METHOD  M_STATE_EXECUTING
VAR_INPUT
END_VAR
VAR_INST
	TargetLayer : INT;
	TargetSlide :E_WareHouseSlide;
END_VAR
VAR
	them: INT;
END_VAR
// Set FB state is busy
Busy := TRUE;

// Process
CASE uiExecutingStep OF
    0: // Command analize
		Ton_BoxMoveForward.IN := FALSE;
		Ton_ArriveDelay.IN := FALSE;
		tonFirstReserveTime.IN :=FALSE;
		tonSecondForwardTime.IN :=FALSE;
		tonThirdReserceTime.IN :=FALSE;
		TargetLayer := WarehouseCoordinates.Layer+(WarehouseSelect-1)*10 ; // Warehouse A=1 , B = 2;
		TargetSlide := WarehouseCoordinates.Slide;
		uiExecutingStep := 10;
		
	10:	//Motor reverse make sure have space can retreat
		Motors.arMotor[TargetLayer].M_MoveBackward();
		Ton_BoxMoveForward.IN := TRUE;
		IF NOT Motors.arMotor[TargetLayer].InStopped  THEN 
			uiExecutingStep := 15;
		END_IF
		IF Ton_BoxMoveForward.Q THEN
			_Error :=TRUE;
			Status :='Storage Cabinet MoveBackward motor timeout';
		END_IF
	15:	//Motor First reverse  then stop motor 
		tonFirstReserveTime.IN := TRUE;
		Ton_BoxMoveForward.IN := FALSE;
		IF tonFirstReserveTime.Q THEN
			tonFirstReserveTime.IN :=FALSE;
			Motors.arMotor[TargetLayer].M_MotorStop();// .M_MotorStop();//('FeedIn Motors.arMotor stop reverse');
			IF Motors.arMotor[TargetLayer].InStopped THEN
				uiExecutingStep := 20;
			END_IF
		END_IF
		
	20:	//Motor SecondForward check cabinet layer have't full box inside 
		Motors.arMotor[TargetLayer].M_MoveForward();// .M_MoveForward();//('FeedIn box : make sure have space can feedIn');
		Ton_BoxMoveForward.IN :=TRUE;
		IF NOT Motors.arMotor[TargetLayer].InStopped THEN
			uiExecutingStep := 25;
		END_IF
		IF Ton_BoxMoveForward.Q THEN
			_Error :=TRUE;
			Status :='Storage Cabinet MoveForward motor timeout';
		END_IF
		
	25:	//Motor second MoveForward  then stop motor
		tonSecondForwardTime.IN := TRUE;
		Ton_BoxMoveForward.IN := FALSE;
		IF tonSecondForwardTime.Q THEN
			tonSecondForwardTime.IN :=FALSE;
			Motors.arMotor[TargetLayer].M_MotorStop();//('');
			IF Motors.arMotor[TargetLayer].InStopped THEN
				uiExecutingStep :=30;
			END_IF
		END_IF
		
	30:	//check layer haven't full box behind
		M_CheckSlideSensor(WarehouseSelect := WarehouseSelect, 
						   WarehouseCoordinates := WarehouseCoordinates,
						   SensorStatus=>CurrentTargetSensorStatus);
		IF NOT  CurrentTargetSensorStatus THEN
			uiExecutingStep :=50;
		ELSE
			_Error :=TRUE;
			Status :='Storage Cabinet Layer full box inside ,plaease remove box ';
		END_IF	
		
	50:
        Motors.arMotor[TargetLayer].M_MoveBackward();// .M_MoveBackward();// ('FeedIn box : conveyor move backward');
		Ton_BoxMoveForward.IN := TRUE;
		IF  NOT Motors.arMotor[TargetLayer].InStopped THEN
			Ton_BoxMoveForward.IN := FALSE;	
			uiExecutingStep := 100;
		END_IF		
		IF  Ton_BoxMoveForward.Q THEN
		  _Error := TRUE;
           Status := 'Move motor timeout';
		END_IF
		
    100: // Wait box arrived
		M_CheckSlideSensor(WarehouseSelect := WarehouseSelect, 
						   WarehouseCoordinates := WarehouseCoordinates,
						   SensorStatus=>CurrentTargetSensorStatus);
        IF NOT CurrentTargetSensorStatus THEN
            uiExecutingStep := 200;
        END_IF
    200:// third reverse 
        tonThirdReserceTime.IN := TRUE;
        IF tonThirdReserceTime.Q THEN
			tonThirdReserceTime.IN :=FALSE;
            uiExecutingStep := 300;
        END_IF
    300:
        Motors.arMotor[TargetLayer].M_MotorStop();//('FeedIn box : conveyor stop move');
        uiExecutingStep := 9900;
    9900:
        // Command completed
        _Executed := TRUE;
END_CASE

IF _Executed THEN
    eState := STATE_DONE;
ELSIF NOT Execute THEN
    eState := STATE_RESETTING;
ELSIF _Error THEN
    eState := STATE_ERROR;
END_IF
END_METHOD

METHOD  M_STATE_RESETTING
VAR_INPUT
END_VAR
VAR 
	uiMotorIndex : UINT;
END_VAR
Done := _Executed;

FOR uiMotorIndex := 1 TO 20 DO 
	Motors.arMotor[uiMotorIndex].M_MotorStop();
END_FOR	
IF NOT Execute THEN
	eState := STATE_DORMANT;
END_IF
END_METHOD

END_FUNCTION_BLOCK

// ---- Library/20_MachineUnits/21_StorageArea/Service/FB_ReloadRoundBeltBoxWithRobot.TcPOU
FUNCTION_BLOCK FB_ReloadRoundBeltBoxWithRobot EXTENDS FB_ObjectBase_V2 IMPLEMENTS IBasicElement
VAR_INPUT
    // Below are the components being controlled.
    Robot         : REFERENCE TO FB_FanucRobot_Basic; // Fanuc Robot
    //AllocatedArea : REFERENCE TO FB_AllocatingSpace; // Allocated area , use to control round belt
	RoundBelt	: REFERENCE TO FB_RoundBeltService;
    WareHouse     : REFERENCE TO FB_WareHouse; // Storage area warehouse A and warehouse B conveyor and sensor
    //	A2_Sensor : REFERENCE TO FB_Sensor;
    //	A3_Sensor : REFERENCE TO FB_Sensor;
	Input : ST_InputTable;
    Info : ST_ReloadRoundBeltBox_Info; // Setting the feedin emptybox action's parameter
    Stop : BOOL;
END_VAR
VAR_OUTPUT
END_VAR
VAR
    strStatus         : STRING;
    tonTimeOut        : TON;
    tonFeedBoxTimeout : TON;
    _UniqueErrorCode  : STRING;
    PreviousStrStatus : STRING;
    PreviousErrorCode : STRING;
    A2_Sensor         : BOOL;
    A3_Sensor         : BOOL;

END_VAR

SUPER^.A10_StateControl();
A2_Sensor := Input.bRoundBelt_ChangeZoneA2Detect_Sensor;
A3_Sensor := Input.bRoundBelt_ChangeZoneA3Detect_Sensor;

ACTION A00_BasicUnits:
tonTimeOut(PT:=T#60S);
tonFeedBoxTimeout(PT:=T#15s);
END_ACTION

METHOD M_CheckCommand : BOOL
VAR_INPUT
END_VAR
VAR_INST
	CheckBehavior : BOOL; // True :Behavior is correct
END_VAR
VAR
	I: INT;
END_VAR
// Memory clear
CheckBehavior := FALSE;
// Check command is correct
IF info.ClampA_Setting.Behavior = E_ClampWork.Work OR info.ClampB_Setting.Behavior = E_ClampWork.Work THEN
	CheckBehavior := TRUE;
ELSE
	CheckBehavior := FALSE;
END_IF


M_CheckCommand := CheckBehavior;
END_METHOD

METHOD M_CheckUnitsNotBusy : BOOL
VAR_INPUT
END_VAR
M_CheckUnitsNotBusy := true;
END_METHOD

METHOD M_CheckUnitsReady : BOOL
VAR_INPUT
END_VAR
M_CheckUnitsReady := true;
END_METHOD

METHOD M_SelectActionMode : E_ReloadRoundBoxAction
VAR_INPUT
END_VAR
IF info.ClampA_Setting.Behavior <> E_ClampWork.Work AND info.ClampB_Setting.Behavior <> E_ClampWork.Work THEN
	M_SelectActionMode :=E_ReloadRoundBoxAction.Undefined;
ELSIF info.ClampA_Setting.Behavior = E_ClampWork.Work AND info.ClampB_Setting.Behavior <> E_ClampWork.Work THEN
	IF info.ClampA_Setting.PickUpArea = E_ReloadRoundBelt_PickupArea.WareHouseA THEN
		M_SelectActionMode := E_ReloadRoundBoxAction.ClampA_WareHouseA;
	ELSIF info.ClampA_Setting.PickUpArea = E_ReloadRoundBelt_PickupArea.WareHouseB THEN
		M_SelectActionMode := E_ReloadRoundBoxAction.ClampA_WareHouseB;
	END_IF
ELSIF info.ClampA_Setting.Behavior <> E_ClampWork.Work AND info.ClampB_Setting.Behavior = E_ClampWork.Work THEN
	IF info.ClampB_Setting.PickUpArea = E_ReloadRoundBelt_PickupArea.WareHouseA THEN
		M_SelectActionMode := E_ReloadRoundBoxAction.ClampB_WareHouseA;
	ELSIF info.ClampB_Setting.PickUpArea = E_ReloadRoundBelt_PickupArea.WareHouseB THEN
		M_SelectActionMode := E_ReloadRoundBoxAction.ClampB_WareHouseB;
	END_IF
ELSIF info.ClampA_Setting.Behavior = E_ClampWork.Work AND info.ClampB_Setting.Behavior = E_ClampWork.Work THEN
	IF info.ClampA_Setting.PickUpArea = E_ReloadRoundBelt_PickupArea.WareHouseA THEN
		IF info.ClampB_Setting.PickUpArea = E_ReloadRoundBelt_PickupArea.WareHouseA THEN
			M_SelectActionMode := E_ReloadRoundBoxAction.A_WareHouseA_B_WareHouseA;
		ELSIF info.ClampB_Setting.PickUpArea = E_ReloadRoundBelt_PickupArea.WareHouseB THEN
			M_SelectActionMode := E_ReloadRoundBoxAction.A_WareHouseA_B_WareHouseB;
		END_IF
	ELSIF info.ClampA_Setting.PickUpArea = E_ReloadRoundBelt_PickupArea.WareHouseB THEN
		IF info.ClampB_Setting.PickUpArea = E_ReloadRoundBelt_PickupArea.WareHouseA THEN
			M_SelectActionMode := E_ReloadRoundBoxAction.A_WareHouseB_B_WareHouseA;
		ELSIF info.ClampB_Setting.PickUpArea = E_ReloadRoundBelt_PickupArea.WareHouseB THEN
			M_SelectActionMode := E_ReloadRoundBoxAction.A_WareHouseB_B_WareHouseB;
		END_IF
	END_IF
END_IF
END_METHOD

METHOD  M_STATE_ABORTED
VAR_INPUT
END_VAR
Busy    := FALSE;
Aborted := TRUE;
UniqueErrorCode:=_UniqueErrorCode;
Status :=strStatus;
IF Reset AND NOT Abort THEN
    eState := STATE_RESETTING;
END_IF
END_METHOD

METHOD  M_STATE_ABORTING
VAR_INPUT
END_VAR
_AbortCompleted := TRUE;
IF _AbortCompleted THEN
    eState := STATE_Aborted;
END_IF
END_METHOD

METHOD  M_STATE_DONE
VAR_INPUT
END_VAR
Busy := FALSE;
Done := TRUE;
IF NOT Execute THEN
    eState := STATE_RESETTING;
END_IF
END_METHOD

METHOD  M_STATE_DORMANT
VAR_INPUT
END_VAR
// Clear FB output
Busy            := FALSE;
Done            := FALSE;
Aborted         := FALSE;
Error           := FALSE;
ErrorID         := 0;
Status          := '';
_ResetCompleted := FALSE;
_Error          := FALSE;
_Executed       := FALSE;
uiExecutingStep := 0;
uiResettingStep := 0;
tonTimeOut.IN:=FALSE;
tonFeedBoxTimeout.IN:=FALSE;
PreviousStrStatus			 :='';
PreviousErrorCode			 :='';
_UniqueErrorCode :='0';
// Wait Execute command
IF Execute THEN
    eState := STATE_EXECUTING;
END_IF
END_METHOD

METHOD  M_STATE_ERROR
VAR_INPUT
END_VAR
UniqueErrorCode:=_UniqueErrorCode;
IF NOT Execute THEN
    eState := STATE_RESETTING;
END_IF
END_METHOD

METHOD M_STATE_EXECUTING
VAR_INPUT
END_VAR
VAR_INST
    ActionMode       : E_ReloadRoundBoxAction;
	BoxReady_1st : BOOL;
	BoxReady_2nd : BOOL;
    CarrierReady_1st : BOOL;
    CarrierReady_2nd : BOOL;
    uiPickUpBothStep : UINT;
    uiPlaceBothStep  : UINT;
    ClampA_WareHouseCoordinates : ST_WareHouseCoordinates;
    ClampB_WareHouseCoordinates : ST_WareHouseCoordinates;
	
	//=============== test only====
		_A2Sensor	:BOOL;
		_A3Sensor	:BOOL;
END_VAR
// Set status busy
Busy := TRUE;
IF THIS^.Stop THEN // Pending the timeout when Stop signal occur
	tonTimeout.IN :=FALSE;
END_IF
CASE uiExecutingStep OF
    0:
        // Clear variable
        ActionMode       := E_ReloadRoundBoxAction.Undefined;
        CarrierReady_1st := FALSE;
        CarrierReady_2nd := FALSE;
        uiPickUpBothStep := 0;
        uiPlaceBothStep  := 0;
		BoxReady_1st := 0;
		BoxReady_2nd := 0;
        // Check command
        IF M_CheckCommand() THEN
            uiExecutingStep := 10;
        END_IF
    10:
        // Start process, check units first
        IF M_CheckUnitsReady() THEN
            uiExecutingStep := 20;
        END_IF
    20:
        // CHeck units not busy state
        IF M_CheckUnitsNotBusy() THEN
            uiExecutingStep := 1000;
        END_IF
    1000:
        // Select action mode
        ActionMode      := M_SelectActionMode();
        uiExecutingStep := 1100;
    1100:
		//DAS_CoreSys.MachineControl.fbAllocateArea.M_ActiveRoundBeltInternalCtrl(); //Request round belt 
		DAS_CoreSys.MachineControl.fbAllocateArea.M_GetRoundBeltAccess(ControlAccess := E_RoundBeltControlAccess.FanucRobot);
        CASE ActionMode OF
            E_ReloadRoundBoxAction.ClampA_WareHouseA:
                uiExecutingStep := 10000;
            E_ReloadRoundBoxAction.ClampA_WareHouseB:
                uiExecutingStep := 11000;
            E_ReloadRoundBoxAction.ClampB_WareHouseA:
                uiExecutingStep := 20000;
            E_ReloadRoundBoxAction.ClampB_WareHouseB:
                uiExecutingStep := 21000;
            E_ReloadRoundBoxAction.A_WareHouseA_B_WareHouseA:
                uiExecutingStep := 30000;
            E_ReloadRoundBoxAction.A_WareHouseA_B_WareHouseB:
                uiExecutingStep := 31000;
            E_ReloadRoundBoxAction.A_WareHouseB_B_WareHouseA:
                uiExecutingStep := 32000;
            E_ReloadRoundBoxAction.A_WareHouseB_B_WareHouseB:
                uiExecutingStep := 33000;
        END_CASE
    10000: // Only ClampA pickup box from WarehouseA
        IF NOT Robot._DI1.Done THEN
            // Read ClampA Warehouse coordinate
            ClampA_WareHouseCoordinates := info.ClampA_Setting.WareHouseSetting;
            // Reload Warehouse target position box
            WareHouse.M_StartReloadBox(WareHouseSelect := E_WareHouse.WareHouseA, WarehouseCoordinates := ClampA_WareHouseCoordinates);

            // Check Box reload completed
            IF WareHouse.bReloadBox_Completed THEN
                BoxReady_1st := TRUE;
            END_IF

            // Robot Warehouse move
            Robot.M_StartWareHousePickUpBox_ClampA(WareHouseSelect := E_WareHouse.WareHouseA,
                                                   Info            := ClampA_WareHouseCoordinates,
                                                   BoxReady_1st    := BoxReady_1st);

            DAS_CoreSys.MachineControl.fbAllocateArea.M_GetRoundBeltAccess(ControlAccess := E_RoundBeltControlAccess.FanucRobot);
            DAS_CoreSys.MachineControl.fbAllocateArea.M_StartReloadRoundBeltAtion(ReloadStation := info.ClampA_Setting.RoundBeltSetting.Station);
        ELSE
			tonTimeOut.IN :=FALSE;
            uiExecutingStep := 10080;
        END_IF
		tonTimeOut.IN :=TRUE;
		IF tonTimeOut.Q THEN
			_Error :=TRUE;
			tonTimeOut.IN :=FALSE;
			strStatus :='Pick Box timeout';
		END_IF
    10080:
        Robot.M_ResetAllCommand(); // Clear command and go to place box
		WareHouse.M_ResetReloadBox();
        IF NOT Robot._DI1.Done THEN
            uiExecutingStep := 60000; // only place clampA
        END_IF
    11000: // Only ClampA pickup box from WarehouseB
        IF NOT Robot._DI1.Done THEN
            // Read ClampA Warehouse coordinate
            ClampA_WareHouseCoordinates := info.ClampA_Setting.WareHouseSetting;
            // Reload Warehouse target position box
            WareHouse.M_StartReloadBox(WareHouseSelect := E_WareHouse.WareHouseB, WarehouseCoordinates := ClampA_WareHouseCoordinates);

            // Check Box reload completed
            IF WareHouse.bReloadBox_Completed THEN
                BoxReady_1st := TRUE;
            END_IF

            // Robot Warehouse move
            Robot.M_StartWareHousePickUpBox_ClampA(WareHouseSelect := E_WareHouse.WareHouseB,
                                                   Info            := ClampA_WareHouseCoordinates,
                                                   BoxReady_1st    := BoxReady_1st);

            DAS_CoreSys.MachineControl.fbAllocateArea.M_GetRoundBeltAccess(ControlAccess := E_RoundBeltControlAccess.FanucRobot);
            DAS_CoreSys.MachineControl.fbAllocateArea.M_StartReloadRoundBeltAtion(ReloadStation := info.ClampA_Setting.RoundBeltSetting.Station);

        ELSE
			tonTimeOut.IN :=FALSE;
            uiExecutingStep := 11080;
        END_IF
		tonTimeOut.IN :=TRUE;
		IF tonTimeOut.Q THEN
			_Error :=TRUE;
			tonTimeOut.IN :=FALSE;
			strStatus :='Pick Box timeout';
		END_IF
    11080:
        Robot.M_ResetAllCommand(); // Clear command and go to place box

        IF NOT Robot._DI1.Done THEN
            uiExecutingStep := 60000; // only place clampA
        END_IF
    20000: // Only ClampB pickup from WarehouseA
        IF NOT Robot._DI1.Done THEN
            // Read ClampA Warehouse coordinate
            ClampB_WareHouseCoordinates := info.ClampB_Setting.WareHouseSetting;
            // Reload Warehouse target position box
            WareHouse.M_StartReloadBox(WareHouseSelect := E_WareHouse.WareHouseA, WarehouseCoordinates := ClampB_WareHouseCoordinates);

            // Check Box reload completed
            IF WareHouse.bReloadBox_Completed THEN
                BoxReady_2nd := TRUE;
            END_IF

            // Robot Warehouse move
            Robot.M_StartWareHousePickUpBox_ClampB(WareHouseSelect := E_WareHouse.WareHouseA,
                                                   Info            := ClampB_WareHouseCoordinates,
                                                   BoxReady_2nd    := BoxReady_2nd);

          	DAS_CoreSys.MachineControl.fbAllocateArea.M_GetRoundBeltAccess(ControlAccess := E_RoundBeltControlAccess.FanucRobot);
            DAS_CoreSys.MachineControl.fbAllocateArea.M_StartReloadRoundBeltAtion(ReloadStation := info.ClampB_Setting.RoundBeltSetting.Station);

        ELSE
			tonTimeOut.IN :=FALSE;
            uiExecutingStep := 20080;
        END_IF
			tonTimeOut.IN :=TRUE;
		IF tonTimeOut.Q THEN
			_Error :=TRUE;
			tonTimeOut.IN :=FALSE;
			strStatus :='Pick Box timeout';
		END_IF
    20080:
        WareHouse.M_ResetReloadBox();
        Robot.M_ResetAllCommand();

        IF NOT Robot._DI1.Done THEN
            uiExecutingStep := 70000; // Only ClampB place box
        END_IF
    21000: // Only ClampB pickup from WarehouseB
        IF NOT Robot._DI1.Done THEN
            // Read ClampA Warehouse coordinate
            ClampB_WareHouseCoordinates := info.ClampB_Setting.WareHouseSetting;
            // Reload Warehouse target position box
            WareHouse.M_StartReloadBox(WareHouseSelect := E_WareHouse.WareHouseB, WarehouseCoordinates := ClampB_WareHouseCoordinates);

            // Check Box reload completed
            IF WareHouse.bReloadBox_Completed THEN
                BoxReady_2nd := TRUE;
            END_IF

            // Robot Warehouse move
            Robot.M_StartWareHousePickUpBox_ClampB(WareHouseSelect := E_WareHouse.WareHouseB,
                                                   Info            := ClampB_WareHouseCoordinates,
                                                   BoxReady_2nd    := BoxReady_2nd);
            DAS_CoreSys.MachineControl.fbAllocateArea.M_GetRoundBeltAccess(ControlAccess := E_RoundBeltControlAccess.FanucRobot);
            DAS_CoreSys.MachineControl.fbAllocateArea.M_StartReloadRoundBeltAtion(ReloadStation := info.ClampA_Setting.RoundBeltSetting.Station);

        ELSE
			tonTimeOut.IN :=FALSE;
            uiExecutingStep := 21080;
        END_IF
			tonTimeOut.IN :=TRUE;
		IF tonTimeOut.Q THEN
			_Error :=TRUE;
			tonTimeOut.IN :=FALSE;
			strStatus :='Pick Box timeout';
		END_IF
    21080:
        WareHouse.M_ResetReloadBox();
        Robot.M_ResetAllCommand();

        IF NOT Robot._DI1.Done THEN
            uiExecutingStep := 70000; // Only ClampB place box
        END_IF
    30000: // ClampA and ClampB pickup box from WarehouseA
        ClampA_WareHouseCoordinates := info.ClampA_Setting.WareHouseSetting;
        ClampB_WareHouseCoordinates := info.ClampB_Setting.WareHouseSetting;

        CASE uiPickUpBothStep OF
            0: // ClampA target slide move the box to front side
                WareHouse.M_StartReloadBox(WareHouseSelect      := E_WareHouse.WareHouseA,
                                           WarehouseCoordinates := ClampA_WareHouseCoordinates);

              	DAS_CoreSys.MachineControl.fbAllocateArea.M_GetRoundBeltAccess(ControlAccess := E_RoundBeltControlAccess.FanucRobot);
                DAS_CoreSys.MachineControl.fbAllocateArea.M_StartReloadRoundBeltAtion(ReloadStation := info.ClampA_Setting.RoundBeltSetting.Station);

                IF WareHouse.bReloadBox_Completed THEN
                    BoxReady_1st     := TRUE;
                    uiPickUpBothStep := 10;
                END_IF

            10: // wait Robot Allow continue
                IF Robot._DI1.Notification AND
                    NOT
                    WareHouse._stWarehouseList.ASide_Layers[ClampA_WareHouseCoordinates.Layer].stStatus.bSlides[ClampA_WareHouseCoordinates.Slide]
                    THEN
                    WareHouse.M_ResetReloadBox();

                    IF NOT WareHouse.bReloadBox_Completed THEN
                        uiPickUpBothStep := 20;
                    END_IF

                END_IF
            20: // ClampB target slide move the box to front slide
                WareHouse.M_StartReloadBox(WareHouseSelect := E_WareHouse.WareHouseA, WarehouseCoordinates := ClampB_WareHouseCoordinates);

                IF WareHouse.bReloadBox_Completed THEN
                    BoxReady_2nd     := TRUE;
                    uiPickUpBothStep := 99;
                END_IF
            99:
        // wait reset
        END_CASE

        Robot.M_StartWareHousePickUpBox_ClampBoth(WareHouseSelect := E_WareHouse.WareHouseA,
                                                  ClampA_Info     := ClampA_WareHouseCoordinates,
                                                  ClampB_Info     := ClampB_WareHouseCoordinates,
                                                  BoxReady_1st    := BoxReady_1st,
                                                  BoxReady_2nd    := BoxReady_2nd);

        IF Robot._DI1.Done THEN
			tonTimeOut.IN :=FALSE;
            uiExecutingStep := 30080;
        END_IF
			tonTimeOut.IN :=TRUE;
		IF tonTimeOut.Q THEN
			_Error :=TRUE;
			tonTimeOut.IN :=FALSE;
			strStatus :='Pick Box timeout';
		END_IF
    30080: // Check robot command is clear
        WareHouse.M_ResetReloadBox();
        Robot.M_ResetAllCommand();

        IF NOT Robot._DI1.Done THEN
            uiExecutingStep := 80000; // go to place step
        END_IF
    31000: // ClampA pickup from Warehouse A, ClampB pickup from Warehouse B
        IF NOT Robot._DI1.Done THEN
            ClampA_WareHouseCoordinates := info.ClampA_Setting.WareHouseSetting;
            WareHouse.M_StartReloadBox(WareHouseSelect := E_WareHouse.WareHouseA, WarehouseCoordinates := ClampA_WareHouseCoordinates);

            IF WareHouse.bReloadBox_Completed THEN
                BoxReady_1st := TRUE;
            END_IF
			DAS_CoreSys.MachineControl.fbAllocateArea.M_ActiveRoundBeltInternalCtrl();
			DAS_CoreSys.MachineControl.fbAllocateArea.M_StartReloadRoundBeltAtion(ReloadStation := info.ClampA_Setting.RoundBeltSetting.Station);
            Robot.M_StartWareHousePickUpBox_ClampA(WareHouseSelect := E_WareHouse.WareHouseA,
                                                   Info            := ClampA_WareHouseCoordinates,
                                                   BoxReady_1st    := BoxReady_1st);
        ELSE
			tonTimeOut.IN :=FALSE;
            uiExecutingStep := 31080;
        END_IF
			tonTimeOut.IN :=TRUE;
		IF tonTimeOut.Q THEN
			_Error :=TRUE;
			tonTimeOut.IN :=FALSE;
			strStatus :='Pick Box timeout';
		END_IF
		
    31080:
        Robot.M_ResetAllCommand(); // Clear command and go to place box
		WareHouse.M_ResetReloadBox();
        IF NOT Robot._di1.Done THEN
            uiExecutingStep := 31100; // ClampA pickup finished, ClampB pickup start
        END_IF
    31100:
        IF NOT Robot._di1.Done THEN
            ClampB_WareHouseCoordinates := info.ClampB_Setting.WareHouseSetting;
            WareHouse.M_StartReloadBox(WareHouseSelect := E_WareHouse.WareHouseB, WarehouseCoordinates := ClampB_WareHouseCoordinates);

            IF WareHouse.bReloadBox_Completed THEN
                BoxReady_2nd := TRUE;
            END_IF

            Robot.M_StartWareHousePickUpBox_ClampB(WareHouseSelect := E_WareHouse.WareHouseB,
                                                   Info            := ClampB_WareHouseCoordinates,
                                                   BoxReady_2nd    := BoxReady_2nd);
        ELSE
			tonTimeOut.IN :=FALSE;
            uiExecutingStep := 31180;
        END_IF
				tonTimeOut.IN :=TRUE;
		IF tonTimeOut.Q THEN
			_Error :=TRUE;
			tonTimeOut.IN :=FALSE;
			strStatus :='Pick Box timeout';
		END_IF
    31180:
        Robot.M_ResetAllCommand(); // Clear command and go to place box

        IF NOT Robot._DI1.Done THEN
            uiExecutingStep := 80000; // only place clampA
        END_IF
    32000: // CLampA pickup from Warehouse B, ClampB pickup from Warehouse A
        IF NOT Robot._DI1.Done THEN
            ClampA_WareHouseCoordinates := info.ClampA_Setting.WareHouseSetting;
            WareHouse.M_StartReloadBox(WareHouseSelect := E_WareHouse.WareHouseB, WarehouseCoordinates := ClampA_WareHouseCoordinates);

            IF WareHouse.bReloadBox_Completed THEN
                BoxReady_1st := TRUE;
            END_IF
            DAS_CoreSys.MachineControl.fbAllocateArea.M_GetRoundBeltAccess(ControlAccess := E_RoundBeltControlAccess.FanucRobot);
            DAS_CoreSys.MachineControl.fbAllocateArea.M_StartReloadRoundBeltAtion(ReloadStation := info.ClampA_Setting.RoundBeltSetting.Station);
            Robot.M_StartWareHousePickUpBox_ClampA(WareHouseSelect := E_WareHouse.WareHouseB,
                                                   Info            := ClampA_WareHouseCoordinates,
                                                   BoxReady_1st    := BoxReady_1st);
        ELSE
			tonTimeOut.IN :=FALSE;
            uiExecutingStep := 32080;
        END_IF
				tonTimeOut.IN :=TRUE;
		IF tonTimeOut.Q THEN
			_Error :=TRUE;
			tonTimeOut.IN :=FALSE;
			strStatus :='Pick Box timeout';
		END_IF
		
    32080:
        Robot.M_ResetAllCommand(); // Clear command and go to place box
		WareHouse.M_ResetReloadBox();
        IF NOT Robot._di1.Done THEN
            uiExecutingStep := 32100; // ClampA pickup finished, ClampB pickup start
        END_IF
    32100:
        IF NOT Robot._di1.Done THEN
            ClampB_WareHouseCoordinates := info.ClampB_Setting.WareHouseSetting;
            WareHouse.M_StartReloadBox(WareHouseSelect := E_WareHouse.WareHouseA, WarehouseCoordinates := ClampB_WareHouseCoordinates);

            IF WareHouse.bReloadBox_Completed THEN
                BoxReady_2nd := TRUE;
            END_IF

            Robot.M_StartWareHousePickUpBox_ClampB(WareHouseSelect := E_WareHouse.WareHouseA,
                                                   Info            := ClampB_WareHouseCoordinates,
                                                   BoxReady_2nd    := BoxReady_2nd);
        ELSE
			tonTimeOut.IN :=FALSE;
            uiExecutingStep := 32180;
        END_IF
				tonTimeOut.IN :=TRUE;
		IF tonTimeOut.Q THEN
			_Error :=TRUE;
			tonTimeOut.IN :=FALSE;
			strStatus :='Pick Box timeout';
		END_IF
		
    32180:
        Robot.M_ResetAllCommand(); // Clear command and go to place box
		WareHouse.M_ResetReloadBox();
        IF NOT Robot._DI1.Done THEN
            uiExecutingStep := 80000; // only place clampA
        END_IF
    33000: // Both Clamp pickup from WarehouseB
        ClampA_WareHouseCoordinates := info.ClampA_Setting.WareHouseSetting;
        ClampB_WareHouseCoordinates := info.ClampB_Setting.WareHouseSetting;

        CASE uiPickUpBothStep OF
            0: // ClampA target slide move the box to front side
                WareHouse.M_StartReloadBox(WareHouseSelect      := E_WareHouse.WareHouseB,
                                           WarehouseCoordinates := ClampA_WareHouseCoordinates);

                DAS_CoreSys.MachineControl.fbAllocateArea.M_GetRoundBeltAccess(ControlAccess := E_RoundBeltControlAccess.FanucRobot );
                DAS_CoreSys.MachineControl.fbAllocateArea.M_StartReloadRoundBeltAtion(ReloadStation := info.ClampA_Setting.RoundBeltSetting.Station);

                IF WareHouse.bReloadBox_Completed THEN
                    BoxReady_1st     := TRUE;
                    uiPickUpBothStep := 10;
                END_IF

            10: // wait Robot Allow continue
                IF Robot._DI1.Notification AND
                    NOT
                    WareHouse._stWarehouseList.BSide_Layers[ClampA_WareHouseCoordinates.Layer].stStatus.bSlides[ClampA_WareHouseCoordinates.Slide]
                    THEN
                    WareHouse.M_ResetReloadBox();

                    IF NOT WareHouse.bReloadBox_Completed THEN
                        uiPickUpBothStep := 20;
                    END_IF

                END_IF
            20: // ClampB target slide move the box to front slide
                WareHouse.M_StartReloadBox(WareHouseSelect := E_WareHouse.WareHouseB, WarehouseCoordinates := ClampB_WareHouseCoordinates);

                IF WareHouse.bReloadBox_Completed THEN
                    BoxReady_2nd     := TRUE;
                    uiPickUpBothStep := 99;
                END_IF
            99:
        // wait reset
        END_CASE

        Robot.M_StartWareHousePickUpBox_ClampBoth(WareHouseSelect := E_WareHouse.WareHouseB,
                                                  ClampA_Info     := ClampA_WareHouseCoordinates,
                                                  ClampB_Info     := ClampB_WareHouseCoordinates,
                                                  BoxReady_1st    := BoxReady_1st,
                                                  BoxReady_2nd    := BoxReady_2nd);

        IF Robot._DI1.Done THEN
			tonTimeOut.IN :=FALSE;
            uiExecutingStep := 33080;
        END_IF
		
			tonTimeOut.IN :=TRUE;
		IF tonTimeOut.Q THEN
			_Error :=TRUE;
			tonTimeOut.IN :=FALSE;
			strStatus :='Pick Box timeout';
		END_IF
		
    33080:
        WareHouse.M_ResetReloadBox();
        Robot.M_ResetAllCommand();

        IF NOT Robot._DI1.Done THEN
            uiExecutingStep := 80000;
        END_IF
    60000: // Only ClampA place box
        WareHouse.M_ResetReloadBox();
        Robot.M_ResetAllCommand();

        // Check Robot RSR1 not working
        IF NOT Robot._di1.Done AND
            NOT (Robot._DI1.AbsMoveA OR
            Robot._DI1.AbsMoveB OR
            Robot._DI1.WarehouseA OR
            Robot._DI1.WarehouseB) THEN
			DAS_CoreSys.MachineControl.fbAllocateArea.M_GetRoundBeltAccess(ControlAccess := E_RoundBeltControlAccess.FanucRobot);
            uiExecutingStep := 61000;
        END_IF
    61000:
        
				DAS_CoreSys.MachineControl.fbAllocateArea.M_GetRoundBeltAccess(ControlAccess := E_RoundBeltControlAccess.FanucRobot);
				DAS_CoreSys.MachineControl.fbAllocateArea.M_StartReloadRoundBeltAtion(ReloadStation := info.ClampA_Setting.RoundBeltSetting.Station);
				IF RoundBelt.xDone  AND arAxisCtrl_gb[AxisNo.RoundBelt].Admin.Axis.Status.NotMoving THEN	
					DAS_CoreSys.MachineControl.fbAllocateArea.M_ResetReloadRoundBeltAction();	
					CarrierReady_1st:=TRUE;			
				 	uiExecutingStep := 61010;
			    END_IF
				IF RoundBelt.xError THEN
					_Error :=TRUE;
					DAS_CoreSys.MachineControl.fbAllocateArea.M_ResetReloadRoundBeltAction();	
					strStatus:='RoundBelt Error';
				END_IF
	61010:
			
        IF NOT Robot._DI1.Done THEN
            Robot.M_StartMoveBoxToRoundBelt_ClampA(CarrierSelect := info.ClampA_Setting.RoundBeltSetting.ReloadCarrier,
                                                   A2_Sensor     := A2_Sensor,
                                                   A3_Sensor     := A3_Sensor,
                                                   RoundBeltSafe := CarrierReady_1st);
        ELSE
			tonTimeOut.IN :=FALSE;
            uiExecutingStep := 61080;
        END_IF
			tonTimeOut.IN :=TRUE;
		IF tonTimeOut.Q THEN
			_Error :=TRUE;
			tonTimeOut.IN :=FALSE;
			strStatus :='Place Box timeout';
		END_IF
		
    61080:
		DAS_CoreSys.MachineControl.fbAllocateArea.M_ResetReloadRoundBeltAction();
        DAS_CoreSys.MachineControl.fbAllocateArea.M_ReleaseRoundBeltAccess(ControlAccess := E_RoundBeltControlAccess.FanucRobot);
        Robot.M_ResetAllCommand();

        IF NOT Robot._DI1.Done THEN
            uiExecutingStep := 99000; // Go to process end
        END_IF
    70000: // Only ClampB place box
        WareHouse.M_ResetReloadBox();
        Robot.M_ResetAllCommand();

        // Check Robot RSR1 not working
        IF NOT Robot._di1.Done AND
            NOT (Robot._DI1.AbsMoveA OR
            Robot._DI1.AbsMoveB OR
            Robot._DI1.WarehouseA OR
            Robot._DI1.WarehouseB) THEN
            uiExecutingStep := 71000;
        END_IF
    71000:
        // Active RoundBelt INTERNAL control
//               DAS_CoreSys.MachineControl.fbAllocateArea.M_GetRoundBeltAccess(ControlAccess := E_RoundBeltControlAccess.FanucRobot);
//               DAS_CoreSys.MachineControl.fbAllocateArea.M_StartReloadRoundBeltAtion(ReloadStation := info.ClampB_Setting.RoundBeltSetting.Station);
				IF RoundBelt.xDone THEN
					DAS_CoreSys.MachineControl.fbAllocateArea.M_ResetReloadRoundBeltAction();
					//DAS_CoreSys.MachineControl.fbAllocateArea.M_ReleaseRoundBeltAccess(ControlAccess := E_RoundBeltControlAccess.FanucRobot);
					CarrierReady_2nd :=TRUE;
				 	uiExecutingStep := 71010;
			    END_IF
				IF RoundBelt.xError THEN
					_Error :=TRUE;
					DAS_CoreSys.MachineControl.fbAllocateArea.M_ResetReloadRoundBeltAction();
					DAS_CoreSys.MachineControl.fbAllocateArea.M_ReleaseRoundBeltAccess(ControlAccess := E_RoundBeltControlAccess.FanucRobot);
					strStatus:='RoundBelt Error';
				END_IF
	71010:
			
        IF NOT Robot._DI1.Done THEN
            Robot.M_StartMoveBoxToRoundBelt_ClampB(CarrierSelect := info.ClampB_Setting.RoundBeltSetting.ReloadCarrier,
                                                   A2_Sensor     := A2_Sensor,
                                                   A3_Sensor     := A3_Sensor,
                                                   RoundBeltSafe := CarrierReady_2nd);
        ELSE
			tonTimeOut.IN :=FALSE;
            uiExecutingStep := 71080;
        END_IF
			tonTimeOut.IN :=TRUE;
		IF tonTimeOut.Q THEN
			_Error :=TRUE;
			tonTimeOut.IN :=FALSE;
			strStatus :='Place Box timeout';
		END_IF
		
    71080:
		DAS_CoreSys.MachineControl.fbAllocateArea.M_ResetReloadRoundBeltAction();
        DAS_CoreSys.MachineControl.fbAllocateArea.M_ReleaseRoundBeltAccess(ControlAccess :=E_RoundBeltControlAccess.FanucRobot );       
        Robot.M_ResetAllCommand();

        IF NOT Robot._DI1.Done THEN
            uiExecutingStep := 99000; // Go to process end
        END_IF
    80000:                            // Both Clamp place box
        WareHouse.M_ResetReloadBox(); // Clear Warehouse reload command
        Robot.M_ResetAllCommand();    // Clear Fanuc Robot command
        IF NOT Robot._DI1.Done THEN
            uiExecutingStep := 81000;
        END_IF;
    81000:
        CASE uiPlaceBothStep OF
            0:
				//=============
				_A2Sensor:=FALSE;
				_A3Sensor:=FALSE;
				//==============
                CarrierReady_1st := FALSE;
                CarrierReady_2nd := FALSE;
				DAS_CoreSys.MachineControl.fbAllocateArea.M_GetRoundBeltAccess(ControlAccess := E_RoundBeltControlAccess.FanucRobot);
                uiPlaceBothStep  := 10;
            10:
                // Check move Round Belt done
                IF RoundBelt.xDone THEN
					DAS_CoreSys.MachineControl.fbAllocateArea.M_ResetReloadRoundBeltAction();
					DAS_CoreSys.MachineControl.fbAllocateArea.M_ReleaseRoundBeltAccess(ControlAccess :=E_RoundBeltControlAccess.FanucRobot );       
                    CarrierReady_1st := TRUE;
                    uiPlaceBothStep  := 11;
                END_IF
				IF RoundBelt.xError THEN
					_Error :=TRUE;
					DAS_CoreSys.MachineControl.fbAllocateArea.M_ResetReloadRoundBeltAction();
					DAS_CoreSys.MachineControl.fbAllocateArea.M_ReleaseRoundBeltAccess(ControlAccess :=E_RoundBeltControlAccess.FanucRobot );       
					strStatus:='RoundBelt Error';
				END_IF
            11:
				//========================Test==================
				IF info.ClampA_Setting.RoundBeltSetting.ReloadCarrier = E_ReloadRoundBelt_PlaceAddress.A2 THEN
					_A2Sensor:=A2_Sensor;
				END_IF
				IF info.ClampA_Setting.RoundBeltSetting.ReloadCarrier = E_ReloadRoundBelt_PlaceAddress.A3 THEN
					_A3Sensor:=A3_Sensor;
				END_IF
				//======================End_test==================
                IF ((info.ClampA_Setting.RoundBeltSetting.ReloadCarrier = E_ReloadRoundBelt_PlaceAddress.A2) AND A2_Sensor) OR
                    ((info.ClampA_Setting.RoundBeltSetting.ReloadCarrier = E_ReloadRoundBelt_PlaceAddress.A3) AND A3_Sensor)
                    THEN
					DAS_CoreSys.MachineControl.fbAllocateArea.M_GetRoundBeltAccess(ControlAccess := E_RoundBeltControlAccess.FanucRobot);
                    uiPlaceBothStep :=20;// 30;
                END_IF
            20:
                // Wait Notification
                IF robot._DI1.Notification THEN
					//========================Test==================
						IF info.ClampA_Setting.RoundBeltSetting.ReloadCarrier = E_ReloadRoundBelt_PlaceAddress.A2 THEN
							_A2Sensor:=FALSE;
						END_IF
						IF info.ClampA_Setting.RoundBeltSetting.ReloadCarrier = E_ReloadRoundBelt_PlaceAddress.A3 THEN
							_A3Sensor:=FALSE;
						END_IF
				//======================End_test==================
                    DAS_CoreSys.MachineControl.fbAllocateArea.M_ResetReloadRoundBeltAction();

                    IF NOT RoundBelt.xDone THEN
                        uiPlaceBothStep := 30;
                    END_IF
                END_IF
            30: // Move Round belt 2nd time
				DAS_CoreSys.MachineControl.fbAllocateArea.M_GetRoundBeltAccess(ControlAccess := E_RoundBeltControlAccess.FanucRobot);
				DAS_CoreSys.MachineControl.fbAllocateArea.M_StartReloadRoundBeltAtion(ReloadStation := info.ClampA_Setting.RoundBeltSetting.Station);
                uiPlaceBothStep := 40;
            40:
                IF RoundBelt.xDone THEN
					DAS_CoreSys.MachineControl.fbAllocateArea.M_ResetReloadRoundBeltAction();
                    CarrierReady_2nd := TRUE;
                    uiPlaceBothStep  := 99;
                END_IF
				IF RoundBelt.xError THEN
					_Error :=TRUE;
					DAS_CoreSys.MachineControl.fbAllocateArea.M_ResetReloadRoundBeltAction();	
					strStatus:='RoundBelt Error';
				END_IF
            99:	
				//========================Test==================
				IF info.ClampB_Setting.RoundBeltSetting.ReloadCarrier = E_ReloadRoundBelt_PlaceAddress.A2 THEN
					_A2Sensor:=A2_Sensor;
				END_IF
				IF info.ClampB_Setting.RoundBeltSetting.ReloadCarrier = E_ReloadRoundBelt_PlaceAddress.A3 THEN
					_A3Sensor:=A3_Sensor;
				END_IF
				//======================End_test==================
        // wait reset
        END_CASE

        IF NOT Robot._DI1.Done THEN
            Robot.M_StartMoveBoxToRoundBelt_Both(CarrierSelect_ClampA := info.ClampA_Setting.RoundBeltSetting.ReloadCarrier,
                                                 CarrierSelect_ClampB := info.ClampB_Setting.RoundBeltSetting.ReloadCarrier,
                                                 A2_Sensor            := _A2Sensor,//A2_Sensor,
                                                 A3_Sensor            := _A3Sensor,//A3_Sensor,
                                                 RoundBeltSafe_1st    := CarrierReady_1st,
                                                 RoundBeltSafe_2nd    := CarrierReady_2nd);
        ELSE
			tonTimeOut.IN :=FALSE;
            uiExecutingStep := 99000;
        END_IF
			tonTimeOut.IN :=TRUE;
		IF tonTimeOut.Q THEN
			_Error :=TRUE;
			tonTimeOut.IN :=FALSE;
			strStatus :='Place Box timeout';
		END_IF
    99000: // process done
        // Stop FeedIn conveyor
					DAS_CoreSys.MachineControl.fbAllocateArea.M_ResetReloadRoundBeltAction();
					DAS_CoreSys.MachineControl.fbAllocateArea.M_ReleaseRoundBeltAccess(ControlAccess :=E_RoundBeltControlAccess.FanucRobot );       
        Status    := 'Process completed';
        _Executed := TRUE;
END_CASE

IF _Executed THEN
    eState := STATE_DONE;
ELSIF NOT Execute THEN
    eState := STATE_RESETTING;
ELSIF Abort THEN
	//FUN_UniqueErrorCodeGenerator(iErrorID := ErrorID,UinqueErrorCode=>_UniqueErrorCode);
	eState :=STATE_ABORTING;
ELSIF _Error THEN
	//FUN_UniqueErrorCodeGenerator(iErrorID := ErrorID,UinqueErrorCode=>_UniqueErrorCode);
	eState :=STATE_ERROR;
END_IF
END_METHOD

METHOD  M_STATE_RESETTING
VAR_INPUT
END_VAR
IF _Executed THEN Done :=TRUE; END_IF

CASE uiResettingStep OF
	0:
					DAS_CoreSys.MachineControl.fbAllocateArea.M_ResetReloadRoundBeltAction();
					DAS_CoreSys.MachineControl.fbAllocateArea.M_ReleaseRoundBeltAccess(ControlAccess :=E_RoundBeltControlAccess.FanucRobot );       
					WareHouse.M_ResetReloadBox();
		Robot.M_ResetAllCommand();
		uiResettingStep := 100;
	100:
		_ResetCompleted := TRUE;
END_CASE
IF _ResetCompleted THEN
    eState := STATE_DORMANT;
END_IF
END_METHOD

END_FUNCTION_BLOCK

// ---- Library/20_MachineUnits/21_StorageArea/Service/FB_RobotRegionMove_AllocatedConveyor.TcPOU
FUNCTION_BLOCK FB_RobotRegionMove_AllocatedConveyor EXTENDS FB_ObjectBase_V2 IMPLEMENTS IBasicElement
VAR_INPUT
    Robot     					: REFERENCE TO FB_FanucRobot_Basic;
	DifferenceCV 				: REFERENCE TO FB_motor;    // Allocated area feed in conveyor(diff and same size conveyor)
	SamesizeCV					: REFERENCE TO FB_motor;
//	SameSizeFullSensor 			: REFERENCE TO BOOL; 				 // Because the same size sensor implement FB_ConveyorSameSize, so use reference to connect it
   // Command   : ST_WareHouseWithRobotMove_Command;
   	cylinder : REFERENCE TO UNI_CylinderList;
   	Input : ST_InputTable;
    Info	  : ST_RobotRegionMove_Info;
	Stop	  : BOOL;
END_VAR
VAR_OUTPUT
  // Status : ST_WareHouseWithRobotMove_Status;
END_VAR
VAR
	_Abort		: BOOL;
	strStatus	: STRING;
	uiResumeStep : UINT;
	
	Area	: E_RobotArea :=E_RobotArea.TransmitCV;
	UseA 	: BOOL;
	UseB	: BOOL;
	SameSizeFullSensor 			: BOOL; 				 // Because the same size sensor implement FB_ConveyorSameSize, so use reference to connect it
	Get 	:BOOL;
	tonTimeOut	:TON;
	tonDelay	:TON;
	tonDelay_SameSizeGetBox : TON;
	tonDelay_SameSizeDelayBox : TON;
	tonFeedBoxTimeout : TON;
	_UniqueErrorCode :STRING;
	PreviousStrStatus : STRING;
	PreviousErrorCode : STRING;
END_VAR


SUPER^.A10_StateControl();
A00_BasicUnits();
SameSizeFullSensor := Input.bSameSizeCV_BoxNearStorageSensor;

ACTION A00_BasicUnits:
tonTimeOut(PT:=T#60S);
tonFeedBoxTimeout(PT:=T#30s);
tonDelay(PT:=T#1.5S);
tonDelay_SameSizeDelayBox(PT:=T#1.5S);
tonDelay_SameSizeGetBox(PT:=T#50MS);
ErrorID:=2210;
END_ACTION

METHOD M_CheckCommand : BOOL // True : Command is useful
VAR_INPUT
END_VAR
VAR
	
END_VAR
// Check command paremeter is correct
	
	THIS^.Get :=Info.Get;	
	UseA :=Info.UseA;
	UseB :=Info.UseB;
	
//Allocated/Empty conveyor
		IF UseA AND ( Info.A_Position<1 OR  Info.A_Position>2 ) THEN
			strStatus:='Wrong command ,Position A Not allow';
			M_CheckCommand:=FALSE;
			RETURN;		
		END_IF
	
		IF UseB AND ( Info.B_Position<1 OR  Info.B_Position>2 )THEN
			strStatus:='Wrong command ,Position B Not allow';
			M_CheckCommand:=FALSE;
			RETURN;		
		END_IF	
M_CheckCommand:=TRUE;
END_METHOD

METHOD M_CheckUnitsNotBusy : BOOL
VAR_INPUT
END_VAR
M_CheckUnitsNotBusy := true;
END_METHOD

METHOD M_CheckUnitsReady : BOOL
VAR_INPUT
END_VAR
M_CheckUnitsReady := true;
END_METHOD

METHOD  M_STATE_ABORTED
VAR_INPUT
END_VAR
ERROR :=TRUE;
Busy    := FALSE;
Aborted := TRUE;
Status := strStatus;
UniqueErrorCode:=_UniqueErrorCode;
_AbortCompleted:=FALSE;
IF NOT Execute THEN
	eSTATE:=STATE_RESETTING;
END_IF

IF Execute AND Reset THEN
	uiExecutingStep :=uiResumeStep;
	PreviousStrStatus := strStatus;
	PreviousErrorCode := _UniqueErrorCode;
	eSTATE:=STATE_EXECUTING;
END_IF
END_METHOD

METHOD  M_STATE_ABORTING
VAR_INPUT
END_VAR
CASE uiAbortingStep OF
	0 :
		uiAbortingStep:=9999;
		tonFeedBoxTimeout.IN :=FALSE;
		tonTimeOut.IN :=FALSE;
		tonDelay.IN :=FALSE;
		_Abort :=FALSE;
		DifferenceCV.M_MotorStop();
		SamesizeCV.M_MotorStop();
		IF strStatus = PreviousStrStatus THEN
			_UniqueErrorCode :=PreviousErrorCode;
		END_IF
		
	9999:	_AbortCompleted:=TRUE;
END_CASE

IF _AbortCompleted THEN	
	eSTATE :=STATE_ABORTED;
END_IF
END_METHOD

METHOD  M_STATE_DONE
VAR_INPUT
END_VAR
Busy := FALSE;
Done := TRUE;
IF NOT Execute THEN
    eState := STATE_RESETTING;
END_IF
END_METHOD

METHOD  M_STATE_DORMANT
VAR_INPUT
END_VAR
// Clear FB output
Busy            := FALSE;
Done            := FALSE;
Aborted         := FALSE;
Error           := FALSE;
ErrorID         := 0;
Status          := '';
_ResetCompleted := FALSE;
_Error          := FALSE;
_Executed       := FALSE;
tonDelay_SameSizeGetBox.IN := FALSE;
tonDelay_SameSizeDelayBox.IN :=false;
tonTimeOut.IN:=FALSE;
strStatus :='No Error';
uiExecutingStep :=uiResettingStep :=uiResumeStep :=0;
tonDelay.IN :=FALSE;
tonFeedBoxTimeout.IN :=FALSE;
_UniqueErrorCode :='0';
PreviousStrStatus			 :='';
PreviousErrorCode			 :='';
// Wait Execute command
IF Execute THEN
    eState := STATE_EXECUTING;
END_IF
END_METHOD

METHOD  M_STATE_ERROR
VAR_INPUT
END_VAR
ERROR   :=TRUE;
Busy	:=FALSE;
Status := strStatus;
UniqueErrorCode:=_UniqueErrorCode;
cylinder.List.fbSameSizeCV_Press3.M_Retract();
cylinder.List.fbSameSizeCV_Press4.M_Retract();
IF NOT Execute THEN	
eSTATE:=STATE_RESETTING;
END_IF
END_METHOD

METHOD  M_STATE_EXECUTING
VAR_INPUT
END_VAR
VAR_INST
	BoxReady_1st : BOOL;
	BoxReady_2nd : BOOL;
    uiBothStep : UINT;
    uiSingleClampStep : UINT;	
	Address_A : INT;
	Address_B : INT;
	bGetBoxInSameSizeConveyor : BOOL;
	uiSameGetBoxStep : UINT;
	bSameSizeCVMoveForward  : BOOL;
	bSameSizeCVMoveBackward : BOOL;
	bDiffCVMoveForward		:BOOL;
	bDiffCVMoveBackward		:BOOL;


END_VAR
VAR
	WareHouse: INT;
	
END_VAR
// Set Busy active edit by johnson
Busy := TRUE;
IF THIS^.Stop THEN // Pending the timeout when Stop signal occur
	tonTimeout.IN :=FALSE;
END_IF

IF bSameSizeCVMoveForward THEN
	IF NOT SamesizeCV.InBackWard THEN
		SamesizeCV.M_MoveForward();
	END_IF
END_IF
IF bSameSizeCVMoveBackward THEN
	IF NOT SamesizeCV.InForWard THEN
	 SamesizeCV.M_MoveBackward();
	END_IF
END_IF
IF bDiffCVMoveForward THEN
	IF NOT DifferenceCV.InBackWard THEN
		DifferenceCV.M_MoveForward();
	END_IF
END_IF
IF bDiffCVMoveBackward THEN
	IF NOT DifferenceCV.InForWard THEN
		DifferenceCV.M_MoveBackward();
	END_IF
END_IF


// Service Process
CASE uiExecutingStep OF
	0:
        // Clear variable
        uiBothStep := 0;
		uiSingleClampStep :=0;
		BoxReady_1st := 0;
		BoxReady_2nd := 0;
		tonTimeOut.IN:=FALSE;
		bSameSizeCVMoveForward  :=FALSE;
		bSameSizeCVMoveBackward :=FALSE;
		bDiffCVMoveForward		:=FALSE;
		bDiffCVMoveBackward		:=FALSE;
        // Check command
        IF M_CheckCommand() THEN
            uiExecutingStep := 10;
		ELSE
			_Error:=TRUE;
        END_IF
    10:
        // Start process, check units first
        IF M_CheckUnitsReady() THEN
            uiExecutingStep := 20;
        END_IF
    20:
        // CHeck units not busy state
        IF M_CheckUnitsNotBusy() THEN
            uiExecutingStep := 1000;
        END_IF
   
	1000:   
			// Read   coordinate
			 Area := THIS^.Area;
 			 Address_A := LREAL_TO_INT(Info.A_Position);
			 Address_B := LREAL_TO_INT(Info.B_Position);
			 bGetBoxInSameSizeConveyor := Get AND ((UseA AND Address_A=2) OR (UseB AND Address_B=2));
			 IF bGetBoxInSameSizeConveyor THEN
				 cylinder.List.fbSameSizeCV_Press3.M_Retract();
				 cylinder.List.fbSameSizeCV_Press4.M_Retract();
			 END_IF
			 uiSameGetBoxStep :=0;
			 tonDelay_SameSizeGetBox.IN:=FALSE;
			IF UseA AND NOT UseB THEN
				//Only clampA
				uiExecutingStep := 10000;
			ELSIF NOT UseA AND UseB THEN
				//Only ClampB 
				uiExecutingStep := 20000;
			ELSIF UseA AND UseB THEN
				//Both Clamps
				uiExecutingStep := 30000;		
			END_IF
       
    10000: // Only ClampA 
        IF NOT Robot._DI1.Done THEN
            
            
			CASE uiSingleClampStep OF
				
				0://
					 IF Get THEN // Get box job
//						IF FeedInConveyor.P_PermitCommand AND NOT FeedInConveyor.P_isRunningBackward THEN
//            				FeedInConveyor.M_AutoMoveReverse(sRecordSource := '');
//						END_IF
//						IF 
					 	
						CASE Address_A OF
							1:
								tonDelay.IN :=Input.bDifferentSizeCV_BoxDetect7_Sensor;
								bDiffCVMoveBackward:=TRUE;
								bDiffCVMoveForward:=FALSE;
								DifferenceCV.M_MoveBackward();
								
							2:
								CASE uiSameGetBoxStep OF
									0:
									//tonDelay.IN :=SameSizeFullSensor;	
									bSameSizeCVMoveBackward := TRUE;
									bSameSizeCVMoveForward := FALSE;
									SamesizeCV.M_MoveBackward();
									cylinder.List.fbSameSizeCV_Press3.M_Retract();
									cylinder.List.fbSameSizeCV_Press4.M_Retract();
									uiSameGetBoxStep :=100;
									
									100:
										tonDelay_SameSizeGetBox.IN := Input.bSameSizeCV_BoxDetect6_Sensor;
										IF tonDelay_SameSizeGetBox.Q THEN
											cylinder.List.fbSameSizeCV_Press3.M_Extend();
											uiSameGetBoxStep :=200;
										END_IF
									200:
										tonDelay_SameSizeGetBox.IN:=FALSE;
										tonDelay_SameSizeDelayBox.IN :=SameSizeFullSensor;
										IF 	tonDelay_SameSizeDelayBox.Q THEN
											uiSameGetBoxStep :=300;
										END_IF	
									300:
										cylinder.List.fbSameSizeCV_Press4.M_Extend();
										tonDelay.IN :=TRUE;
										uiSameGetBoxStep :=400;
									400: 
										IF tonDelay.Q THEN
											cylinder.List.fbSameSizeCV_Press4.M_Retract();
										END_IF
								END_CASE
						END_CASE	
			
					ELSE
//						IF FeedInConveyor.P_PermitCommand AND NOT FeedInConveyor.P_isRunningBackward THEN
//            				FeedInConveyor.M_MoveForward(sRecordSource := '');
//						END_IF
						CASE Address_A OF
							1:
								tonDelay.IN := NOT Input.bDifferentSizeCV_BoxDetect7_Sensor;
								bDiffCVMoveForward :=TRUE;
								bDiffCVMoveBackward:=FALSE;
								DifferenceCV.M_MoveForward();
							2:
								tonDelay.IN :=NOT SameSizeFullSensor;
								bSameSizeCVMoveForward :=TRUE;
								bSameSizeCVMoveBackward:=FALSE;
								SamesizeCV.M_MoveForward();			
						END_CASE					
				
					END_IF	
				
						IF tonDelay.Q THEN
							tonFeedBoxTimeout.IN :=FALSE;
							uiSingleClampStep:=1000;
						END_IF
						tonFeedBoxTimeout.IN :=TRUE;
						IF tonFeedBoxTimeout.Q THEN
							tonFeedBoxTimeout.IN :=FALSE;
							strStatus :='Feed Box timeout';
							uiResumeStep:=10000;
							_Abort:=TRUE;
						END_IF
				1000:
						BoxReady_1st:=TRUE;
						tonDelay.IN:=FALSE;
						bSameSizeCVMoveForward  :=FALSE;
						bSameSizeCVMoveBackward :=FALSE;
						bDiffCVMoveForward		:=FALSE;
						bDiffCVMoveBackward		:=FALSE;						
						DifferenceCV.M_MotorStop();
						SamesizeCV.M_MotorStop();
						uiSingleClampStep:=9999;
				9999: //Wait	
			END_CASE
			          		 
				  // Robot Abs move
           		 Robot.M_StartRobotAbsMove(GetBox:=Get,
											UseClampA:=UseA,
											UseClampB:=UseB,
											Area:=Area,
											ClampA_Address:=Address_A,
											ClampB_Address:=Address_B,
											BoxReady_1:=BoxReady_1st,
											BoxReady_2:=BoxReady_2nd);				  
		
        ELSE
			tonTimeOut.IN:=FALSE;
            uiExecutingStep := 10080;
        END_IF
		tonTimeOut.IN:=TRUE;
		IF tonTimeOut.Q=TRUE THEN
			tonTimeOut.IN:=FALSE;
			strStatus :='Robot move timeout';
			_Error:=TRUE;
		END_IF	
    10080:
        Robot.M_ResetRobotAbsMove(UseA,UseB); // Clear command and go to place box
		tonTimeOut.IN:=TRUE;
		uiSameGetBoxStep:=0;
        IF NOT Robot._DI1.Done THEN
			tonTimeOut.IN:=FALSE;
            uiExecutingStep := 50000; 
        END_IF
		
    	IF tonTimeOut.Q=TRUE THEN
			strStatus :='Reset Robot timeout';
			_Error:=TRUE;
		END_IF	
    
   20000: // Only ClampB
        IF NOT Robot._DI1.Done THEN
            			
			CASE uiSingleClampStep OF
			0:	
					 IF Get THEN // Get box job
//						IF FeedInConveyor.P_PermitCommand AND NOT FeedInConveyor.P_isRunningBackward THEN
//            				FeedInConveyor.M_AutoMoveReverse(sRecordSource := '');
//						END_IF
//						IF 
					 	
						CASE Address_B OF
							1:
								tonDelay.IN :=Input.bDifferentSizeCV_BoxDetect7_Sensor;
								bDiffCVMoveBackward:=TRUE;
								bDiffCVMoveForward := FALSE;
								DifferenceCV.M_MoveBackward();
								
							2:
//								tonDelay.IN :=SameSizeFullSensor;	
//								SamesizeCV.M_MoveBackward();
//								cylinder.List.fbSameSizeCV_Press3.M_Retract();
//								cylinder.List.fbSameSizeCV_Press4.M_Retract();
								CASE uiSameGetBoxStep OF
									0:
									//tonDelay.IN :=SameSizeFullSensor;	
									bSameSizeCVMoveForward :=FALSE;
									bSameSizeCVMoveBackward := TRUE;
									SamesizeCV.M_MoveBackward();
									cylinder.List.fbSameSizeCV_Press3.M_Retract();
									cylinder.List.fbSameSizeCV_Press4.M_Retract();
									uiSameGetBoxStep :=100;
									
									100:
										tonDelay_SameSizeGetBox.IN := Input.bSameSizeCV_BoxDetect6_Sensor;
										IF tonDelay_SameSizeGetBox.Q THEN
											cylinder.List.fbSameSizeCV_Press3.M_Extend();
											uiSameGetBoxStep :=200;
										END_IF
									200:
										tonDelay_SameSizeGetBox.IN:=FALSE;
										tonDelay_SameSizeDelayBox.IN :=SameSizeFullSensor;
										IF 	tonDelay_SameSizeDelayBox.Q THEN
											uiSameGetBoxStep :=300;
										END_IF	
									300:
										cylinder.List.fbSameSizeCV_Press4.M_Extend();
										uiSameGetBoxStep :=400;
									400: 
										tonDelay.IN :=TRUE;
										IF tonDelay.Q THEN
											cylinder.List.fbSameSizeCV_Press4.M_Retract();
										END_IF
								END_CASE			

						END_CASE	
			
					ELSE
//						IF FeedInConveyor.P_PermitCommand AND NOT FeedInConveyor.P_isRunningBackward THEN
//            				FeedInConveyor.M_MoveForward(sRecordSource := '');
//						END_IF
						CASE Address_B OF
							1:
								tonDelay.IN := NOT Input.bDifferentSizeCV_BoxDetect7_Sensor;
								bDiffCVMoveForward	:=TRUE;
								bDiffCVMoveBackward	:=FALSE;
								DifferenceCV.M_MoveForward();
							2:
								tonDelay.IN :=NOT SameSizeFullSensor;
								bSameSizeCVMoveForward :=TRUE;
								bSameSizeCVMoveBackward :=FALSE;
								SamesizeCV.M_MoveForward();			
						END_CASE					
				
					END_IF	
				
						IF tonDelay.Q THEN
							tonFeedBoxTimeout.IN :=FALSE;
							uiSingleClampStep:=1000;
						END_IF
						tonFeedBoxTimeout.IN :=TRUE;
						IF tonFeedBoxTimeout.Q THEN
							tonFeedBoxTimeout.IN :=FALSE;
							strStatus :='Feed Box timeout';
							uiResumeStep:=10000;
							_Abort:=TRUE;
						END_IF
				1000:
						//BoxReady_1st:=TRUE;
						BoxReady_2nd:=TRUE;
						tonDelay.IN:=FALSE;
						bSameSizeCVMoveForward  :=FALSE;
						bSameSizeCVMoveBackward :=FALSE;
						bDiffCVMoveForward		:=FALSE;
						bDiffCVMoveBackward		:=FALSE;
						DifferenceCV.M_MotorStop();
						SamesizeCV.M_MotorStop();
						uiSingleClampStep:=9999;
				9999: //Wait	

			END_CASE
			          		 
				  // Robot Abs move
           		 Robot.M_StartRobotAbsMove( GetBox:=Get,
											UseClampA:=UseA,
											UseClampB:=UseB,
											Area:=Area,
											ClampA_Address:=Address_A,
											ClampB_Address:=Address_B,
											BoxReady_1:=BoxReady_1st,
											BoxReady_2:=BoxReady_2nd);	
        ELSE
			tonTimeOut.IN:=FALSE;
            uiExecutingStep := 20080;
        END_IF
		tonTimeOut.IN:=TRUE;
		IF tonTimeOut.Q=TRUE THEN
			tonTimeOut.IN:=FALSE;
			strStatus :='Robot move timeout';
			_Error:=TRUE;
		END_IF	
    20080:
       Robot.M_ResetRobotAbsMove(UseA,UseB);; // Clear command 
		uiSameGetBoxStep :=0;
        IF NOT Robot._DI1.Done THEN
            uiExecutingStep := 50000; 
        END_IF
		tonTimeOut.IN:=TRUE;
		IF tonTimeOut.Q=TRUE THEN
			strStatus :='Reset Robot timeout';
			_Error:=TRUE;
		END_IF	
    30000: // Both Clamps
        		
		
		  CASE uiBothStep OF
           		0://	
					BoxReady_1st := FALSE;
					BoxReady_2nd := FALSE;					
					uiBothStep:=1000;						
				
				1000:
						IF Get THEN // Get box job
							CASE Address_A OF
								1:
									tonDelay.IN :=Input.bDifferentSizeCV_BoxDetect7_Sensor;
									bDiffCVMoveForward	:=FALSE;
									bDiffCVMoveBackward	:=TRUE;
									DifferenceCV.M_MoveBackward();
									
								2:
//									tonDelay.IN :=SameSizeFullSensor;	
//									SamesizeCV.M_MoveBackward();
//									cylinder.List.fbSameSizeCV_Press3.M_Retract();
//									cylinder.List.fbSameSizeCV_Press4.M_Retract();
								CASE uiSameGetBoxStep OF
									0:
									//tonDelay.IN :=SameSizeFullSensor;	
									bSameSizeCVMoveForward  :=FALSE;
									bSameSizeCVMoveBackward :=TRUE;
									SamesizeCV.M_MoveBackward();
									cylinder.List.fbSameSizeCV_Press3.M_Retract();
									cylinder.List.fbSameSizeCV_Press4.M_Retract();
									uiSameGetBoxStep :=100;
									
									100:
										tonDelay_SameSizeGetBox.IN := Input.bSameSizeCV_BoxDetect6_Sensor;
										IF tonDelay_SameSizeGetBox.Q THEN
											cylinder.List.fbSameSizeCV_Press3.M_Extend();
											uiSameGetBoxStep :=200;
										END_IF
									200:
										tonDelay_SameSizeGetBox.IN:=FALSE;
										tonDelay_SameSizeDelayBox.IN :=SameSizeFullSensor;
										IF 	tonDelay_SameSizeDelayBox.Q THEN
											uiSameGetBoxStep :=300;
										END_IF	
									300:
										cylinder.List.fbSameSizeCV_Press4.M_Extend();
										tonDelay.IN :=TRUE;
										uiSameGetBoxStep :=400;
									400: 
										IF tonDelay.Q THEN
											cylinder.List.fbSameSizeCV_Press4.M_Retract();
										END_IF
								END_CASE
				
							END_CASE	
			
						ELSE
							CASE Address_A OF
								1:
									tonDelay.IN := NOT Input.bDifferentSizeCV_BoxDetect7_Sensor;
									bDiffCVMoveForward	:=TRUE;
									bDiffCVMoveBackward	:=FALSE;
									DifferenceCV.M_MoveForward();
								2:
									tonDelay.IN :=NOT SameSizeFullSensor;
									bSameSizeCVMoveForward  :=TRUE;
									bSameSizeCVMoveBackward :=FALSE;
									SamesizeCV.M_MoveForward();			
							END_CASE					
				
						END_IF	
				
						IF tonDelay.Q THEN
							tonFeedBoxTimeout.IN :=FALSE;
							uiSameGetBoxStep:=0;
							uiBothStep:=2000;
						END_IF
						tonFeedBoxTimeout.IN :=TRUE;
						IF tonFeedBoxTimeout.Q THEN
							tonFeedBoxTimeout.IN :=FALSE;
							strStatus :='Feed Box timeout';
							uiResumeStep:=30000;
							_Abort:=TRUE;
						END_IF
				2000:
						tonDelay.IN :=FALSE;
						bSameSizeCVMoveForward  :=FALSE;
						bSameSizeCVMoveBackward :=FALSE;
						bDiffCVMoveForward		:=FALSE;
						bDiffCVMoveBackward		:=FALSE;
						DifferenceCV.M_MotorStop();
						SamesizeCV.M_MotorStop();
						BoxReady_1st:=TRUE;
						tonDelay_SameSizeGetBox.IN := FALSE;
						tonDelay_SameSizeDelayBox.IN :=FALSE;
						IF Robot._DI1.Notification THEN
							uiBothStep:=3000;
						END_IF
				3000:
						IF Get THEN // Get box job
							CASE Address_B OF
								1:
									tonDelay.IN :=Input.bDifferentSizeCV_BoxDetect7_Sensor;
									bDiffCVMoveForward	:=FALSE;
									bDiffCVMoveBackward :=TRUE;
									DifferenceCV.M_MoveBackward();
									
								2:
//									tonDelay.IN :=SameSizeFullSensor;	
//									SamesizeCV.M_MoveBackward();
//									cylinder.List.fbSameSizeCV_Press3.M_Retract();
//									cylinder.List.fbSameSizeCV_Press4.M_Retract();
									CASE uiSameGetBoxStep OF
									0:
									//tonDelay.IN :=SameSizeFullSensor;	
									bSameSizeCVMoveForward :=FALSE;
									bSameSizeCVMoveBackward :=TRUE;
									SamesizeCV.M_MoveBackward();
									cylinder.List.fbSameSizeCV_Press3.M_Retract();
									cylinder.List.fbSameSizeCV_Press4.M_Retract();
									uiSameGetBoxStep :=100;
									
									100:
										tonDelay_SameSizeGetBox.IN := Input.bSameSizeCV_BoxDetect6_Sensor;
										IF tonDelay_SameSizeGetBox.Q THEN
											cylinder.List.fbSameSizeCV_Press3.M_Extend();
											uiSameGetBoxStep :=200;
										END_IF
									200:
										tonDelay_SameSizeGetBox.IN:=FALSE;
										tonDelay_SameSizeDelayBox.IN :=SameSizeFullSensor;
										IF 	tonDelay_SameSizeDelayBox.Q THEN
											uiSameGetBoxStep :=300;
										END_IF	
									300:
										cylinder.List.fbSameSizeCV_Press4.M_Extend();
										tonDelay.IN :=TRUE;
										uiSameGetBoxStep :=400;
									400: 
										IF tonDelay.Q THEN
											cylinder.List.fbSameSizeCV_Press4.M_Retract();
										END_IF
								END_CASE
							END_CASE	
			
						ELSE
							CASE Address_B OF
								1:
									tonDelay.IN := NOT Input.bDifferentSizeCV_BoxDetect7_Sensor;
									bDiffCVMoveForward	:=TRUE;
									bDiffCVMoveBackward := FALSE;
									DifferenceCV.M_MoveForward();
								2:
									tonDelay.IN :=NOT SameSizeFullSensor;
									bSameSizeCVMoveForward :=TRUE;
									bSameSizeCVMoveBackward := FALSE;
									SamesizeCV.M_MoveForward();			
							END_CASE					
				
						END_IF	
				
						IF tonDelay.Q THEN
							tonFeedBoxTimeout.IN :=FALSE;
							uiBothStep:=9000;
						END_IF
						IF tonFeedBoxTimeout.Q THEN
							tonFeedBoxTimeout.IN :=FALSE;
							strStatus :='Feed Box timeout';
							uiResumeStep:=30000;
							_Abort:=TRUE;
						END_IF
				
				9000:
						BoxReady_2nd:=TRUE;
						tonDelay.IN :=FALSE;
						bSameSizeCVMoveForward  :=FALSE;
						bSameSizeCVMoveBackward :=FALSE;
						bDiffCVMoveForward		:=FALSE;
						bDiffCVMoveBackward		:=FALSE;
						DifferenceCV.M_MotorStop();
						SamesizeCV.M_MotorStop();
				
					
       
      	  END_CASE

       	  // Robot Abs move
           		 Robot.M_StartRobotAbsMove( GetBox:=Get,
											UseClampA:=UseA,
											UseClampB:=UseB,
											Area:=Area,
											ClampA_Address:=Address_A,
											ClampB_Address:=Address_B,
											BoxReady_1:=BoxReady_1st,
											BoxReady_2:=BoxReady_2nd);	
		
		
        IF Robot._DI1.Done THEN
			tonTimeOut.IN:=FALSE;
            uiExecutingStep := 30080;
        END_IF
			tonTimeOut.IN:=TRUE;
		IF tonTimeOut.Q=TRUE THEN
			tonTimeOut.IN:=FALSE;
			strStatus :='Robot move timeout';
			_Abort:=TRUE;
		END_IF
    30080: // Check robot command is clear
        
        Robot.M_ResetRobotAbsMove(UseA,UseB);

        IF NOT Robot._DI1.Done THEN
			tonTimeOut.IN:=FALSE;
            uiExecutingStep := 50000; // go to place step
        END_IF    
   		tonTimeOut.IN:=TRUE;
		IF tonTimeOut.Q=TRUE THEN
			strStatus :='Stop Robot timeout';
			_Error:=TRUE;
		END_IF	
  	50000:	// if robot put need box forward more time
			IF NOT Get THEN
				uiExecutingStep :=51000;
			ELSE
				uiExecutingStep :=99000;
			END_IF
    51000:	//conveyor forward 
			IF UseA THEN
				CASE Address_A OF
					1:
						tonDelay.IN := NOT Input.bDifferentSizeCV_BoxDetect7_Sensor;
						DifferenceCV.M_MoveForward();
					2:
						tonDelay.IN :=NOT SameSizeFullSensor;
						SamesizeCV.M_MoveForward();			
				END_CASE
			END_IF					
			IF UseB THEN
				CASE Address_B OF
					1:
						tonDelay.IN := NOT Input.bDifferentSizeCV_BoxDetect7_Sensor;
						DifferenceCV.M_MoveForward();
					2:
						tonDelay.IN :=NOT SameSizeFullSensor;
						SamesizeCV.M_MoveForward();			
				END_CASE
			END_IF
						IF tonDelay.Q THEN
							tonFeedBoxTimeout.IN :=FALSE;
							uiExecutingStep:=99000;
						END_IF
						IF tonFeedBoxTimeout.Q THEN
							tonFeedBoxTimeout.IN :=FALSE;
							strStatus :='Feed Box timeout';
							uiResumeStep:=30000;
							_Abort:=TRUE;
						END_IF
    99000: // process done
         Status    := 'Process completed';
		 bSameSizeCVMoveForward  :=FALSE;
		 bSameSizeCVMoveBackward :=FALSE;
		 bDiffCVMoveForward		:=FALSE;
		 bDiffCVMoveBackward		:=FALSE;
		 cylinder.List.fbSameSizeCV_Press3.M_Retract();
		 cylinder.List.fbSameSizeCV_Press4.M_Retract();
        _Executed := TRUE;
END_CASE
IF _Executed THEN
    eState := STATE_DONE;
ELSIF _Error THEN
	//FUN_UniqueErrorCodeGenerator(iErrorID := ErrorID,UinqueErrorCode=>_UniqueErrorCode);
	eState := STATE_ERROR;
ELSIF NOT Execute THEN
    eState := STATE_RESETTING;
END_IF
IF _Abort OR Abort THEN
	//FUN_UniqueErrorCodeGenerator(iErrorID := ErrorID,UinqueErrorCode=>_UniqueErrorCode);
	eSTATE:=STATE_ABORTING;
END_IF
END_METHOD

METHOD  M_STATE_RESETTING
VAR_INPUT
END_VAR
Error :=FALSE;
Done :=FALSE;
Busy := FALSE;


CASE uiResettingStep OF
	
	0:
		tonTimeOut.IN:=FALSE;
		tonDelay_SameSizeDelayBox.IN :=FALSE;
		Robot.M_ResetAllCommand();
		Robot.M_ResetRobotAbsMove(TRUE,TRUE);
		DifferenceCV.M_MotorStop();
		SamesizeCV.M_MotorStop();
		cylinder.List.fbSameSizeCV_Press3.M_Retract();
		cylinder.List.fbSameSizeCV_Press4.M_Retract();
		uiResettingStep:=100;
		
	100:	
	
		uiResettingStep:=9999;
	9999:
		_ResetCompleted:=TRUE;
END_CASE
IF _ResetCompleted THEN
	eSTATE:=STATE_DORMANT;
END_IF
END_METHOD

END_FUNCTION_BLOCK

// ---- Library/20_MachineUnits/21_StorageArea/Service/FB_RobotRegionMove_BufferArea.TcPOU
FUNCTION_BLOCK FB_RobotRegionMove_BufferArea EXTENDS FB_ObjectBase_V2 IMPLEMENTS IBasicElement
VAR_INPUT
    Robot : REFERENCE TO FB_FanucRobot_Basic;
    // Command   : ST_WareHouseWithRobotMove_Command;
    Info : ST_RobotRegionMove_Info;
    Stop : BOOL;
END_VAR
VAR_OUTPUT
    // Status : ST_WareHouseWithRobotMove_Status;

END_VAR
VAR
    _Abort       : BOOL;
    strStatus    : STRING;
    uiResumeStep : UINT;

    Area : E_RobotArea := E_RobotArea.BufferArea;
    UseA : BOOL;
    UseB : BOOL;

    Get               : BOOL;
    tonTimeOut        : TON;
    _UniqueErrorCode  : STRING;
    PreviousStrStatus : STRING;
    PreviousErrorCode : STRING;
END_VAR

SUPER^.A10_StateControl();
A00_BasicUnits();

METHOD M_CheckCommand : BOOL // True : Command is useful
VAR_INPUT
END_VAR
VAR
	
END_VAR
// Check command paremeter is correct

THIS^.Get :=Info.Get;
UseA := Info.UseA;
UseB := Info.UseB;
//Buffer area
		
		IF UseA AND ( Info.A_Position<1 OR  Info.A_Position>40) THEN
			strStatus:='Wrong command ,Position A Not allow';
			M_CheckCommand:=FALSE;
			RETURN;			
		END_IF		
	
		IF UseB AND( Info.B_Position<1 OR  Info.B_Position>40 )THEN
			strStatus:='Wrong command ,Position B Not allow';
			M_CheckCommand:=FALSE;
			RETURN;			
		END_IF
		
M_CheckCommand:=TRUE;
END_METHOD

METHOD M_CheckUnitsNotBusy : BOOL
VAR_INPUT
END_VAR
M_CheckUnitsNotBusy := true;
END_METHOD

METHOD M_CheckUnitsReady : BOOL
VAR_INPUT
END_VAR
M_CheckUnitsReady := true;
END_METHOD

METHOD  M_STATE_ABORTED
VAR_INPUT
END_VAR
ERROR :=TRUE;
Busy    := FALSE;
Aborted := TRUE;
Status := strStatus;
UniqueErrorCode:=_UniqueErrorCode;
IF NOT Execute THEN
	eSTATE:=STATE_RESETTING;
END_IF

IF Execute AND Reset THEN
	uiExecutingStep :=uiResumeStep;
	PreviousStrStatus := strStatus;
	PreviousErrorCode := _UniqueErrorCode;
	eSTATE:=STATE_EXECUTING;
END_IF
END_METHOD

METHOD  M_STATE_ABORTING
VAR_INPUT
END_VAR
CASE uiAbortingStep OF
	0 :
		uiAbortingStep:=9999;
		IF strStatus = PreviousStrStatus THEN
			_UniqueErrorCode :=PreviousErrorCode;
		END_IF
		_Abort :=FALSE;
	9999:	_AbortCompleted:=TRUE;
END_CASE

IF _AbortCompleted THEN	
	eSTATE :=STATE_ABORTED;
END_IF
END_METHOD

METHOD  M_STATE_DONE
VAR_INPUT
END_VAR
Busy := FALSE;
Done := TRUE;
IF NOT Execute THEN
    eState := STATE_RESETTING;
END_IF
END_METHOD

METHOD  M_STATE_DORMANT
VAR_INPUT
END_VAR
// Clear FB output
Busy            := FALSE;
Done            := FALSE;
Aborted         := FALSE;
Error           := FALSE;
ErrorID         := 0;
Status          := '';
_ResetCompleted := FALSE;
_Error          := FALSE;
_Executed       := FALSE;

tonTimeOut.IN:=FALSE;
strStatus :='No Error';
uiExecutingStep :=uiResettingStep :=uiResumeStep :=0;
PreviousStrStatus			 :='';
PreviousErrorCode			 :='';
_UniqueErrorCode	:='0';

// Wait Execute command
IF Execute THEN
    eState := STATE_EXECUTING;
END_IF
END_METHOD

METHOD  M_STATE_ERROR
VAR_INPUT
END_VAR
ERROR   :=TRUE;
Busy	:=FALSE;
Status := strStatus;
UniqueErrorCode:=_UniqueErrorCode;
IF NOT Execute THEN	
eSTATE:=STATE_RESETTING;
END_IF
END_METHOD

METHOD  M_STATE_EXECUTING
VAR_INPUT
END_VAR
VAR_INST
    ActionMode       : E_ReloadRoundBoxAction;
	BoxReady_1st : BOOL;
	BoxReady_2nd : BOOL;
    CarrierReady_1st : BOOL;
    CarrierReady_2nd : BOOL;
    uiBothStep : UINT;
    uiSingleClampStep : UINT;
	Address_A : INT;
	Address_B : INT;
END_VAR
VAR
	WareHouse: INT;
END_VAR
// Set Busy active edit by johnson
Busy := TRUE;
IF THIS^.Stop THEN // Pending the timeout when Stop signal occur
	tonTimeout.IN :=FALSE;
END_IF
// Service Process
CASE uiExecutingStep OF
	0:
        // Clear variable
        ActionMode       := E_ReloadRoundBoxAction.Undefined;
        CarrierReady_1st := FALSE;
        CarrierReady_2nd := FALSE;
        uiBothStep := 0;
		uiSingleClampStep :=0;
		BoxReady_1st := 0;
		BoxReady_2nd := 0;
		tonTimeOut.IN:=FALSE;
        // Check command
        IF M_CheckCommand() THEN
            uiExecutingStep := 10;
		ELSE
			_Error:=TRUE;
        END_IF
    10:
        // Start process, check units first
        IF M_CheckUnitsReady() THEN
            uiExecutingStep := 20;
        END_IF
    20:
        // CHeck units not busy state
        IF M_CheckUnitsNotBusy() THEN
            uiExecutingStep := 1000;
        END_IF
   
	1000:   
			// Read   coordinate
 			 Address_A := LREAL_TO_INT(Info.A_Position);
			 Address_B := LREAL_TO_INT(Info.B_Position);
			 
			IF UseA AND NOT UseB THEN
				//Only clampA
				uiExecutingStep := 10000;
			ELSIF NOT UseA AND UseB THEN
				//Only ClampB 
				uiExecutingStep := 20000;
			ELSIF UseA AND UseB THEN
				//Both Clamps
				uiExecutingStep := 30000;		
			END_IF
       
    10000: // Only ClampA 
        IF NOT Robot._DI1.Done THEN            
           		BoxReady_1st:=TRUE;				
			          		 
				  // Robot Abs move
           		 Robot.M_StartRobotAbsMove(GetBox:=Get,
											UseClampA:=UseA,
											UseClampB:=UseB,
											Area:=Area,
											ClampA_Address:=Address_A,
											ClampB_Address:=Address_B,
											BoxReady_1:=BoxReady_1st,
											BoxReady_2:=BoxReady_2nd);	  
		
        ELSE
			tonTimeOut.IN:=FALSE;
            uiExecutingStep := 10080;
        END_IF
			tonTimeOut.IN:=TRUE;
			IF tonTimeOut.Q=TRUE THEN
				tonTimeOut.IN:=FALSE;			
				strStatus :='Reset Robot timeout';
				_Error:=TRUE;
			END_IF	
    10080:
        Robot.M_ResetRobotAbsMove(UseA,UseB); // Clear command and go to place box
		tonTimeOut.IN:=TRUE;
        IF NOT Robot._DI1.Done THEN
			tonTimeOut.IN:=FALSE;
            uiExecutingStep := 99000; 
        END_IF
    	IF tonTimeOut.Q=TRUE THEN
			strStatus :='Reset Robot timeout';
			_Error:=TRUE;
		END_IF	
    
   20000: // Only ClampB
        IF NOT Robot._DI1.Done THEN           		
				BoxReady_2nd:=TRUE;				          		 
				  // Robot Abs move
           		 Robot.M_StartRobotAbsMove( GetBox:=Get,
											UseClampA:=UseA,
											UseClampB:=UseB,
											Area:=Area,
											ClampA_Address:=Address_A,
											ClampB_Address:=Address_B,
											BoxReady_1:=BoxReady_1st,
											BoxReady_2:=BoxReady_2nd);	
        ELSE
			tonTimeOut.IN:=FALSE;
            uiExecutingStep := 20080;
        END_IF
		tonTimeOut.IN:=TRUE;
			IF tonTimeOut.Q=TRUE THEN
				tonTimeOut.IN:=FALSE;			
				strStatus :='Reset Robot timeout';
				_Error:=TRUE;
			END_IF	
    20080:
       Robot.M_ResetRobotAbsMove(UseA,UseB);; // Clear command 

        IF NOT Robot._DI1.Done THEN
            uiExecutingStep := 99000; 
        END_IF
		tonTimeOut.IN:=TRUE;
		IF tonTimeOut.Q=TRUE THEN
			strStatus :='Reset Robot timeout';
			_Error:=TRUE;
		END_IF	
    30000: // Both Clamps
        		
		
		  CASE uiBothStep OF
           		0://	
					BoxReady_1st := FALSE;
					BoxReady_2nd := FALSE;					
					uiBothStep:=1000;	
	
				1000:
						BoxReady_1st:=TRUE;
						uiBothStep:=2000;
						
				2000:
						IF Robot._DI1.Notification THEN
							uiBothStep:=3000;
						END_IF
				3000:
					
					
						uiBothStep:=9000;	
					
				9000:
						BoxReady_2nd:=TRUE;
						uiBothStep:=9999;
				
				9999: //Wait		
        // wait reset
        END_CASE

       	  // Robot Abs move
           		 Robot.M_StartRobotAbsMove( GetBox:=Get,
											UseClampA:=UseA,
											UseClampB:=UseB,
											Area:=Area,
											ClampA_Address:=Address_A,
											ClampB_Address:=Address_B,
											BoxReady_1:=BoxReady_1st,
											BoxReady_2:=BoxReady_2nd);	
		
		
        IF Robot._DI1.Done THEN
			tonTimeOut.IN:=FALSE;
            uiExecutingStep := 30080;
        END_IF
		IF tonTimeOut.Q=TRUE THEN
				tonTimeOut.IN:=FALSE;			
				strStatus :='Reset Robot timeout';
				_Error:=TRUE;
			END_IF	
    30080: // Check robot command is clear
        
        Robot.M_ResetRobotAbsMove(UseA,UseB);

        IF NOT Robot._DI1.Done THEN
			tonTimeOut.IN:=FALSE;
            uiExecutingStep := 99000; // go to place step
        END_IF    
   		tonTimeOut.IN:=TRUE;
		IF tonTimeOut.Q=TRUE THEN
			strStatus :='Stop Robot timeout';
			_Error:=TRUE;
		END_IF	
   
    99000: // process done
                Status    := 'Process completed';
        _Executed := TRUE;
END_CASE

IF _Executed THEN
    eState := STATE_DONE;
ELSIF _Error THEN
	//FUN_UniqueErrorCodeGenerator(iErrorID := ErrorID,UinqueErrorCode=>_UniqueErrorCode);
    eState := STATE_ERROR;
ELSIF NOT Execute THEN
    eState := STATE_RESETTING;
END_IF
IF _Abort OR Abort THEN
	//FUN_UniqueErrorCodeGenerator(iErrorID := ErrorID,UinqueErrorCode=>_UniqueErrorCode);
	eSTATE:=STATE_ABORTING;
END_IF
END_METHOD

METHOD  M_STATE_RESETTING
VAR_INPUT
END_VAR
Error :=FALSE;
Done :=FALSE;
Busy := FALSE;


CASE uiResettingStep OF
	
	0:
		tonTimeOut.IN:=FALSE;
		Robot.M_ResetAllCommand();
		Robot.M_ResetRobotAbsMove(TRUE,TRUE);
		
		uiResettingStep:=9999;
	9999:
		_ResetCompleted:=TRUE;
END_CASE
IF _ResetCompleted THEN
	eSTATE:=STATE_DORMANT;
END_IF
END_METHOD

END_FUNCTION_BLOCK

// ---- Library/20_MachineUnits/21_StorageArea/Service/FB_RobotRegionMove_FeedInConveyor.TcPOU
FUNCTION_BLOCK FB_RobotRegionMove_FeedInConveyor EXTENDS FB_ObjectBase_V2 IMPLEMENTS IBasicElement
VAR_INPUT
    Robot     					: REFERENCE TO FB_FanucRobot_Basic;
	LowerConveyor				: REFERENCE TO FB_Motor;
	Input : REFERENCE TO ST_InputTable;

   // Command   : ST_WareHouseWithRobotMove_Command;
    Info	  : ST_RobotRegionMove_Info;
	Stop	  : BOOL;
END_VAR
VAR_OUTPUT
  // Status : ST_WareHouseWithRobotMove_Status;
  
END_VAR
VAR
	_Abort		: BOOL;
	strStatus	: STRING;
	uiResumeStep : UINT;
	
	Area	: E_RobotArea := E_RobotArea.InOutConveyor;
	UseA 	: BOOL;
	UseB	: BOOL;
	
	Get 	:BOOL;
	tonTimeOut	:TON;
	TON_DelayTransMove	:TON;
	_UniqueErrorCode :STRING;
	PreviousStrStatus : STRING;
	PreviousErrorCode : STRING;
END_VAR

SUPER^.A10_StateControl();
A00_BasicUnits();

ACTION A00_BasicUnits:
tonTimeOut(PT:=T#60S);
TON_DelayTransMove(PT :=T#2S);
ErrorID:=2240;
END_ACTION

METHOD M_CheckCommand : BOOL // True : Command is useful
VAR_INPUT
END_VAR
VAR
	
END_VAR
// Check command paremeter is correct
	
	THIS^.Get :=Info.Get;
	UseA := Info.UseA;
	UseB := Info.UseB;

	 //FeedIn/Out conveyor
	 	IF UseA THEN	 
			IF  (Info.A_Position<1 OR  Info.A_Position>3 )THEN
				strStatus:='Wrong command ,Position A Not allow';
				M_CheckCommand:=FALSE;
				RETURN;	
			ELSIF  Info.A_Position=3 AND Get THEN
				strStatus:='Wrong command ,Can Not Get box from FeedOut conveyor ';
				M_CheckCommand:=FALSE;
				RETURN;
			ELSIF 	Info.A_Position <>3 AND NOT Get THEN
				strStatus:='Wrong command ,Can Not Put box to FeedIn conveyor ';
				M_CheckCommand:=FALSE;
				RETURN;				
			END_IF
		END_IF
		
		IF UseB AND ( Info.B_Position<1 OR  Info.B_Position>3 )THEN
			strStatus:='Wrong command ,Position B Not allow';
			M_CheckCommand:=FALSE;
			RETURN;	
		ELSIF UseB AND Info.B_Position=3 AND Get THEN
			strStatus:='Wrong command ,Can Not Get box from FeedOut conveyor ';
			M_CheckCommand:=FALSE;
			RETURN;		
		ELSIF UseB AND Info.B_Position <>3 AND NOT Get THEN
			strStatus:='Wrong command ,Can Not Put box to FeedIn conveyor ';
			M_CheckCommand:=FALSE;
			RETURN;		
		END_IF
		
M_CheckCommand:=TRUE;
END_METHOD

METHOD M_CheckUnitsNotBusy : BOOL
VAR_INPUT
END_VAR
M_CheckUnitsNotBusy := true;
END_METHOD

METHOD M_CheckUnitsReady : BOOL
VAR_INPUT
END_VAR
M_CheckUnitsReady := true;
END_METHOD

METHOD  M_STATE_ABORTED
VAR_INPUT
END_VAR
ERROR :=TRUE;
Busy    := FALSE;
Aborted := TRUE;
Status := strStatus;
UniqueErrorCode:=_UniqueErrorCode;
IF NOT Execute THEN
	eSTATE:=STATE_RESETTING;
END_IF

IF Execute AND Reset THEN
	PreviousStrStatus := strStatus;
	PreviousErrorCode := _UniqueErrorCode;
	uiExecutingStep :=uiResumeStep;
	eSTATE:=STATE_EXECUTING;
END_IF
END_METHOD

METHOD  M_STATE_ABORTING
VAR_INPUT
END_VAR
CASE uiAbortingStep OF
	0 :
		tonTimeOut.IN:=FALSE;
		TON_DelayTransMove.IN :=FALSE;
		LowerConveyor.M_MotorStop();
		IF strStatus = PreviousStrStatus THEN
			_UniqueErrorCode :=PreviousErrorCode;
		END_IF
		uiAbortingStep:=9999;
	
	9999:	_AbortCompleted:=TRUE;
END_CASE

IF _AbortCompleted THEN	
	eSTATE :=STATE_ABORTED;
END_IF
END_METHOD

METHOD  M_STATE_DONE
VAR_INPUT
END_VAR
Busy := FALSE;
Done := TRUE;
IF NOT Execute THEN
    eState := STATE_RESETTING;
END_IF
END_METHOD

METHOD  M_STATE_DORMANT
VAR_INPUT
END_VAR
// Clear FB output
Busy            := FALSE;
Done            := FALSE;
Aborted         := FALSE;
Error           := FALSE;
ErrorID         := 0;
Status          := '';
_ResetCompleted := FALSE;
_Error          := FALSE;
_Executed       := FALSE;

tonTimeOut.IN:=FALSE;
TON_DelayTransMove.IN :=FALSE;
strStatus :='No Error';
uiExecutingStep :=uiResettingStep :=uiResumeStep :=0;
_UniqueErrorCode :='0';
PreviousStrStatus			 :='';
PreviousErrorCode			 :='';

// Wait Execute command
IF Execute THEN
    eState := STATE_EXECUTING;
END_IF
END_METHOD

METHOD  M_STATE_ERROR
VAR_INPUT
END_VAR
ERROR   :=TRUE;
Busy	:=FALSE;
Status := strStatus;
UniqueErrorCode:=_UniqueErrorCode;
IF NOT Execute THEN	
eSTATE:=STATE_RESETTING;
END_IF
END_METHOD

METHOD  M_STATE_EXECUTING
VAR_INPUT
END_VAR
VAR_INST
	BoxReady_1st : BOOL;
	BoxReady_2nd : BOOL;
    uiBothStep : UINT;
    uiSingleClampStep : UINT;	
	Address_A : INT;
	Address_B : INT;
END_VAR
VAR
	WareHouse: INT;
END_VAR
// Set Busy active edit by johnson
Busy := TRUE;
IF THIS^.Stop THEN // Pending the timeout when Stop signal occur
	tonTimeout.IN :=FALSE;
END_IF
// Service Process
CASE uiExecutingStep OF
	0:
        // Clear variable
        uiBothStep := 0;
		uiSingleClampStep :=0;
		BoxReady_1st := 0;
		BoxReady_2nd := 0;
		tonTimeOut.IN:=FALSE;
        // Check command
        IF M_CheckCommand() THEN
            uiExecutingStep := 10;
		ELSE
			_Error:=TRUE;
        END_IF
    10:
        // Start process, check units first
        IF M_CheckUnitsReady() THEN
            uiExecutingStep := 20;
        END_IF
    20:
        // CHeck units not busy state
        IF M_CheckUnitsNotBusy() THEN
            uiExecutingStep := 1000;
        END_IF
   
	1000:   
			// Read   coordinate
			 Area := THIS^.Area;
 			 Address_A := LREAL_TO_INT(Info.A_Position);
			 Address_B := LREAL_TO_INT(Info.B_Position);
			 
			IF UseA AND NOT UseB THEN
				//Only clampA
				uiExecutingStep := 10000;
			ELSIF NOT UseA AND UseB THEN
				//Only ClampB 
				uiExecutingStep := 20000;
			ELSIF UseA AND UseB THEN
				//Both Clamps
				uiExecutingStep := 30000;		
			END_IF
       
    10000: // Only ClampA 
        IF NOT Robot._DI1.Done THEN
            
            
			CASE uiSingleClampStep OF
				
				0://
				
					CASE Address_A OF
						1,2:
							uiSingleClampStep:=1000;
						
						3: 
							uiSingleClampStep:=100;
					END_CASE
				
				100:	
					LowerConveyor.M_MoveBackward();
					IF ( NOT Input.bLowCV_BoxArrived_Sensor) AND ( Input.bLowCV_2ndBoxGap_Sensor) THEN
						tonTimeOut.IN:=FALSE;
						uiSingleClampStep:=200;
					END_IF
					tonTimeOut.IN:=TRUE;
					IF tonTimeOut.Q=TRUE THEN
						strStatus :='Empty Conveyor timeout';
						uiResumeStep:=10000;
						_Abort:=TRUE;
					END_IF
				200:
					TON_DelayTransMove.IN :=TRUE;
					IF TON_DelayTransMove.Q THEN
						LowerConveyor.M_MotorStop();
						uiSingleClampStep:=300;
					END_IF
				
				300:
					TON_DelayTransMove.IN :=FALSE;
					IF 	LowerConveyor.InStopped THEN
						tonTimeOut.IN:=FALSE;
						BoxReady_1st:=TRUE;
						uiSingleClampStep:=9999;
					END_IF
					tonTimeOut.IN:=TRUE;
					IF tonTimeOut.Q=TRUE THEN
						strStatus :='Stop Conveyor timeout';
						_Error:=TRUE;
					END_IF	
				
				1000:
						CASE Address_A OF
							
						1:
							BoxReady_1st:=Input.bUpCV_Block1Detect_Sensor;
						
						2:
							BoxReady_1st:=Input.bUpCV_BoxArrived_Sensor;
						END_CASE						
						
				9999: //
				
			END_CASE
			          		 
				  // Robot Abs move
           		 Robot.M_StartRobotAbsMove(GetBox:=Get,
											UseClampA:=UseA,
											UseClampB:=UseB,
											Area:=Area,
											ClampA_Address:=Address_A,
											ClampB_Address:=Address_B,
											BoxReady_1:=BoxReady_1st,
											BoxReady_2:=BoxReady_2nd);				  
		
        ELSE
			tonTimeOut.IN:=FALSE;
            uiExecutingStep := 10080;
        END_IF
		tonTimeOut.IN:=TRUE;
		IF tonTimeOut.Q=TRUE THEN
			tonTimeOut.IN:=FALSE;
			strStatus :='Reset Robot timeout';
			_Error:=TRUE;
		END_IF	
    10080:
        Robot.M_ResetRobotAbsMove(UseA,UseB); // Clear command and go to place box
		tonTimeOut.IN:=TRUE;
        IF NOT Robot._DI1.Done THEN
			tonTimeOut.IN:=FALSE;
            uiExecutingStep := 80000; 
        END_IF
    	IF tonTimeOut.Q=TRUE THEN
			strStatus :='Reset Robot timeout';
			_Error:=TRUE;
		END_IF	
    
	10090: // Check box 
		
			
   20000: // Only ClampB
        IF NOT Robot._DI1.Done THEN
			
            	CASE uiSingleClampStep OF
				
				0://
				
					CASE Address_B OF
						1,2:
							uiSingleClampStep:=1000;
						
						3: 
							uiSingleClampStep:=100;
					END_CASE
			
				100:	
					LowerConveyor.M_MoveBackward();
					IF (NOT Input.bLowCV_BoxArrived_Sensor) AND  Input.bLowCV_2ndBoxGap_Sensor THEN
						tonTimeOut.IN:=FALSE;
						uiSingleClampStep:=200;
					END_IF
					tonTimeOut.IN:=TRUE;
					IF tonTimeOut.Q=TRUE THEN
						strStatus :='Empty Conveyor timeout';
						uiResumeStep:=20000;
						_Abort:=TRUE;
					END_IF
				200:
					TON_DelayTransMove.IN :=TRUE;
					IF TON_DelayTransMove.Q THEN
						LowerConveyor.M_MotorStop();
						uiSingleClampStep:=300;
					END_IF
				
				300:
					TON_DelayTransMove.IN := FALSE;
					IF 	LowerConveyor.InStopped THEN
						tonTimeOut.IN:=FALSE;
						BoxReady_2nd:=TRUE;
						uiSingleClampStep:=9999;
					END_IF
					tonTimeOut.IN:=TRUE;
					IF tonTimeOut.Q=TRUE THEN
						strStatus :='Stop Conveyor timeout';
						_Error:=TRUE;
					END_IF	
				
				1000:
						CASE Address_B OF
							
						1:
							BoxReady_2nd:=Input.bUpCV_Block1Detect_Sensor;
						
						2:
							BoxReady_2nd:=Input.bUpCV_BoxArrived_Sensor;
						END_CASE						
						
				9999 ://
			END_CASE	
		
			
			          		 
				  // Robot Abs move
           		 Robot.M_StartRobotAbsMove( GetBox:=Get,
											UseClampA:=UseA,
											UseClampB:=UseB,
											Area:=Area,
											ClampA_Address:=Address_A,
											ClampB_Address:=Address_B,
											BoxReady_1:=BoxReady_1st,
											BoxReady_2:=BoxReady_2nd);	
        ELSE
			tonTimeOut.IN:=FALSE;
            uiExecutingStep := 20080;
        END_IF
		tonTimeOut.IN:=TRUE;
		IF tonTimeOut.Q=TRUE THEN
			tonTimeOut.IN:=FALSE;
			strStatus :='Reset Robot timeout';
			_Error:=TRUE;
		END_IF	
    20080:
       Robot.M_ResetRobotAbsMove(UseA,UseB);; // Clear command 

        IF NOT Robot._DI1.Done THEN
            uiExecutingStep := 80000; 
        END_IF
		tonTimeOut.IN:=TRUE;
		IF tonTimeOut.Q=TRUE THEN
			strStatus :='Reset Robot timeout';
			_Error:=TRUE;
		END_IF	
		
	
			
		
    30000: // Both Clamps
        		
		
		  CASE uiBothStep OF
           		0://	
					BoxReady_1st := FALSE;
					BoxReady_2nd := FALSE;
					CASE Address_A OF
						1,2:
							uiBothStep:=1000;
						
						3: 
							uiBothStep:=100;
					END_CASE				
				100:	
					LowerConveyor.M_MoveBackward();
					tonTimeOut.IN:=FALSE;
					IF (NOT Input.bLowCV_BoxArrived_Sensor) AND  Input.bLowCV_2ndBoxGap_Sensor THEN
						uiBothStep:=200;
					END_IF
					tonTimeOut.IN:=TRUE;
					IF tonTimeOut.Q=TRUE THEN
						strStatus :='Empty conveyor timeout';
						uiResumeStep:=30000;
						_Abort:=TRUE;
					END_IF	
				200:
					TON_DelayTransMove.IN := TRUE;
					IF TON_DelayTransMove.Q THEN 
						LowerConveyor.M_MotorStop();
						uiBothStep:=300;
					END_IF
				
				300:
					TON_DelayTransMove.IN :=FALSE;
					IF 	LowerConveyor.InStopped THEN
						tonTimeOut.IN:=FALSE;
						BoxReady_1st:=TRUE;
						uiBothStep:=1000;
					END_IF
					tonTimeOut.IN:=TRUE;
					IF tonTimeOut.Q=TRUE THEN
						strStatus :='Stop conveyor timeout';
						_Error:=TRUE;
					END_IF		
				1000:
				
							CASE Address_A OF							
						1:
							BoxReady_1st:=Input.bUpCV_Block1Detect_Sensor;
						
						2:
							BoxReady_1st:=Input.bUpCV_BoxArrived_Sensor;
						END_CASE
						IF Robot._DI1.Notification THEN
							BoxReady_1st:=TRUE;
							uiBothStep:=2000;
						END_IF
						
						
				2000:
						BoxReady_1st:=TRUE;
						CASE Address_B OF
						1,2:
							uiBothStep:=9000;						
						3: 
							uiBothStep:=3000;
					END_CASE	
				
				3000:	
					LowerConveyor.M_MoveBackward();
					IF (NOT Input.bLowCV_BoxArrived_Sensor) AND Input.bLowCV_2ndBoxGap_Sensor THEN
						tonTimeOut.IN:=FALSE;
						uiBothStep:=3200;
					END_IF
					tonTimeOut.IN:=TRUE;
					IF tonTimeOut.Q=TRUE THEN
						strStatus :='Empty conveyor timeout';
						uiResumeStep:=30000;
						_Abort:=TRUE;
					END_IF	
				3200:
					TON_DelayTransMove.IN := TRUE;
					IF TON_DelayTransMove.Q THEN 
						LowerConveyor.M_MotorStop();
						uiBothStep:=3300;
					END_IF					
				
				3300:
						TON_DelayTransMove.IN :=FALSE;
					IF 	LowerConveyor.InStopped THEN
						tonTimeOut.IN:=FALSE;
						BoxReady_2nd:=TRUE;
						uiBothStep:=9999;
					END_IF
					tonTimeOut.IN:=TRUE;
					IF tonTimeOut.Q=TRUE THEN
						strStatus :='Stop conveyor timeout';
						_Error:=TRUE;
					END_IF		
				9000:
							CASE Address_B OF							
						1:
							BoxReady_2nd:=Input.bUpCV_Block1Detect_Sensor ;
						
						2:
							BoxReady_2nd:=Input.bUpCV_BoxArrived_Sensor;
						END_CASE
				
				9999: //Wait		
        // wait reset
        END_CASE

       	  // Robot Abs move
           		 Robot.M_StartRobotAbsMove( GetBox:=Get,
											UseClampA:=UseA,
											UseClampB:=UseB,
											Area:=Area,
											ClampA_Address:=Address_A,
											ClampB_Address:=Address_B,
											BoxReady_1:=BoxReady_1st,
											BoxReady_2:=BoxReady_2nd);	
		
		
        IF Robot._DI1.Done THEN
			tonTimeOut.IN:=FALSE;
            uiExecutingStep := 30080;
        END_IF
		tonTimeOut.IN:=TRUE;
		IF tonTimeOut.Q=TRUE THEN
			tonTimeOut.IN:=FALSE;
			strStatus :='Reset Robot timeout';
			_Error:=TRUE;
		END_IF
    30080: // Check robot command is clear
        
        Robot.M_ResetRobotAbsMove(UseA,UseB);

        IF NOT Robot._DI1.Done THEN
			tonTimeOut.IN:=FALSE;
            uiExecutingStep := 80000; // go to place step
        END_IF    
   		tonTimeOut.IN:=TRUE;
		IF tonTimeOut.Q=TRUE THEN
			strStatus :='Stop Robot timeout';
			_Error:=TRUE;
		END_IF	
   
		
	80000:
		IF UseA THEN
			CASE Address_A OF
			1:
//				IF Input.bUpCV_BoxArrived_Sensor.P_SignalState THEN
//					strStatus :='Box not taken on F1';
//					_Error:=TRUE;
//				END_IF
				 uiExecutingStep :=99000;
			2:	
//				IF Input.bUpCV_Block1Detect_Sensor.P_SignalState THEN
//					strStatus :='Box not taken on F2';
//					_Error:=TRUE;
//				END_IF	
					uiExecutingStep :=99000;

			3:
				uiExecutingStep :=81000;			
			END_CASE
		END_IF
		IF UseB THEN
			CASE Address_B OF
			1:
//				IF Input.bUpCV_BoxArrived_Sensor.P_SignalState THEN
//					strStatus :='Box not taken on F1';
//					_Error:=TRUE;
//				END_IF
				 uiExecutingStep :=99000;
			2:	
//				IF Input.bUpCV_Block1Detect_Sensor.P_SignalState THEN
//					strStatus :='Box not taken on F2';
//					_Error:=TRUE;
//				END_IF	
					uiExecutingStep :=99000;

			3:
				uiExecutingStep :=81000;			
			END_CASE
		END_IF
		
	81000:
			LowerConveyor.M_MoveBackward();
			tonTimeOut.IN:=FALSE;
			IF (NOT Input.bLowCV_BoxArrived_Sensor) AND ( Input.bLowCV_2ndBoxGap_Sensor) THEN
						uiExecutingStep:=81100;
			END_IF
			tonTimeOut.IN:=TRUE;
			IF tonTimeOut.Q=TRUE THEN
				strStatus :='Empty conveyor timeout';
				_Error:=TRUE;
			END_IF	
	81100:		
			TON_DelayTransMove.IN := TRUE;
			IF TON_DelayTransMove.Q THEN
			LowerConveyor.M_MotorStop();
			uiExecutingStep:=81200;
			END_IF
				
	81200:
			TON_DelayTransMove.IN := false;
			IF 	LowerConveyor.InStopped THEN
				tonTimeOut.IN:=FALSE;
				uiExecutingStep:=99000;
			END_IF
			tonTimeOut.IN:=TRUE;
			IF tonTimeOut.Q=TRUE THEN
				strStatus :='Stop conveyor timeout';
				_Error:=TRUE;
			END_IF		
					
    99000: // process done
          Status    := 'Process completed';
      	  _Executed := TRUE;
END_CASE
IF _Executed THEN
    eState := STATE_DONE;
ELSIF _Error THEN
//	FUN_UniqueErrorCodeGenerator(iErrorID := ErrorID,UinqueErrorCode=>_UniqueErrorCode);
    eState := STATE_ERROR;
ELSIF NOT Execute THEN
    eState := STATE_RESETTING;
END_IF
IF _Abort OR Abort THEN
//	FUN_UniqueErrorCodeGenerator(iErrorID := ErrorID,UinqueErrorCode=>_UniqueErrorCode);
	eSTATE:=STATE_ABORTING;
END_IF
END_METHOD

METHOD  M_STATE_RESETTING
VAR_INPUT
END_VAR
Error :=FALSE;
Done :=FALSE;
Busy := FALSE;


CASE uiResettingStep OF
	
	0:
		tonTimeOut.IN:=FALSE;
		TON_DelayTransMove.IN :=FALSE;
		Robot.M_ResetAllCommand();
		Robot.M_ResetRobotAbsMove(TRUE,TRUE);
		uiResettingStep:=100;
		
	100:
	
		LowerConveyor.M_MotorStop();	
		uiResettingStep:=9999;
	9999:
		_ResetCompleted:=TRUE;
END_CASE
IF _ResetCompleted THEN
	eSTATE:=STATE_DORMANT;
END_IF
END_METHOD

END_FUNCTION_BLOCK

// ---- Library/20_MachineUnits/21_StorageArea/Service/FB_RobotRegionMove_PullOutConveyor.TcPOU
FUNCTION_BLOCK FB_RobotRegionMove_PullOutConveyor EXTENDS FB_ObjectBase_V2 IMPLEMENTS IBasicElement
VAR_INPUT
    Robot     				: REFERENCE TO FB_FanucRobot_Basic;
	PullOutConveyor 		: REFERENCE TO FB_PullOutConveyorAction; // Allocated area pull out conveyor
    Info	  				: ST_RobotRegionMove_Info;
	Stop	  : BOOL;
END_VAR
VAR_OUTPUT
  // Status : ST_WareHouseWithRobotMove_Status;
END_VAR
VAR
	_Abort		: BOOL;
	strStatus	: STRING;
	uiResumeStep : UINT;
	
	Area	: E_RobotArea:=E_RobotArea.PullOutConveyor;
	UseA 	: BOOL;
	UseB	: BOOL;
	
	Get 	:BOOL;
	tonTimeOut	:TON;
	_UniqueErrorCode :STRING;
	PreviousStrStatus : STRING;
	PreviousErrorCode : STRING;
END_VAR

SUPER^.A10_StateControl();
A00_BasicUnits();

ACTION A00_BasicUnits:
tonTimeOut(PT:=T#60S);
ErrorID:=2230;
END_ACTION

METHOD M_CheckCommand : BOOL // True : Command is useful
VAR_INPUT
END_VAR
VAR
	
END_VAR
// Check command paremeter is correct
		
	THIS^.Get :=Info.Get;
	UseA :=Info.UseA;
	UseB :=Info.UseB;

	 // PullOut conveyor
		IF UseA AND (Info.A_Position<1 OR  Info.A_Position>2 )THEN
			strStatus:='Wrong command ,Position A Not allow';
			M_CheckCommand:=FALSE;
			RETURN;				
		END_IF	
	
		IF UseB AND (Info.B_Position<1 OR  Info.B_Position>2 )THEN
			strStatus:='Wrong command ,Position B Not allow';
			M_CheckCommand:=FALSE;
			RETURN;			
		END_IF
	



M_CheckCommand:=TRUE;
END_METHOD

METHOD M_CheckUnitsNotBusy : BOOL
VAR_INPUT
END_VAR
M_CheckUnitsNotBusy := true;
END_METHOD

METHOD M_CheckUnitsReady : BOOL
VAR_INPUT
END_VAR
M_CheckUnitsReady := true;
END_METHOD

METHOD  M_STATE_ABORTED
VAR_INPUT
END_VAR
ERROR :=TRUE;
Busy    := FALSE;
Aborted := TRUE;
Status := strStatus;
UniqueErrorCode:=_UniqueErrorCode;
IF NOT Execute THEN
	eSTATE:=STATE_RESETTING;
END_IF

IF Execute AND Reset THEN
	PreviousStrStatus := strStatus;
	PreviousErrorCode := _UniqueErrorCode;
	uiExecutingStep :=uiResumeStep;
	eSTATE:=STATE_EXECUTING;
END_IF
END_METHOD

METHOD  M_STATE_ABORTING
VAR_INPUT
END_VAR
CASE uiAbortingStep OF
	0 :
		uiAbortingStep:=9999;
		DAS_CoreSys.MachineControl.fbStorageArea.M_ResetSlides_FeedOut();
		tonTimeOut.IN:=FALSE;
		_Abort :=FALSE;
		IF strStatus = PreviousStrStatus THEN
			_UniqueErrorCode :=PreviousErrorCode;
		END_IF
	9999:	_AbortCompleted:=TRUE;
END_CASE

IF _AbortCompleted THEN	
	eSTATE :=STATE_ABORTED;
END_IF
END_METHOD

METHOD  M_STATE_DONE
VAR_INPUT
END_VAR
Busy := FALSE;
Done := TRUE;
IF NOT Execute THEN
    eState := STATE_RESETTING;
END_IF
END_METHOD

METHOD  M_STATE_DORMANT
VAR_INPUT
END_VAR
// Clear FB output
Busy            := FALSE;
Done            := FALSE;
Aborted         := FALSE;
Error           := FALSE;
ErrorID         := 0;
Status          := '';
_ResetCompleted := FALSE;
_Error          := FALSE;
_Executed       := FALSE;

tonTimeOut.IN:=FALSE;
strStatus :='No Error';
uiExecutingStep :=uiResettingStep :=uiResumeStep :=0;
PreviousStrStatus			 :='';
PreviousErrorCode			 :='';

// Wait Execute command
IF Execute THEN
    eState := STATE_EXECUTING;
END_IF
END_METHOD

METHOD  M_STATE_ERROR
VAR_INPUT
END_VAR
ERROR   :=TRUE;
Busy	:=FALSE;
Status := strStatus;
UniqueErrorCode:=_UniqueErrorCode;
IF NOT Execute THEN	
eSTATE:=STATE_RESETTING;
END_IF
END_METHOD

METHOD  M_STATE_EXECUTING
VAR_INPUT
END_VAR
VAR_INST
	BoxReady_1st : BOOL;
	BoxReady_2nd : BOOL;
    uiBothStep : UINT;
    uiSingleClampStep : UINT;	
	Area : E_RobotArea;
	Address_A : INT;
	Address_B : INT;
END_VAR
VAR
	WareHouse: INT;
	LowerConveyor: INT;
END_VAR
// Set Busy active edit by johnson
Busy := TRUE;

IF THIS^.Stop THEN // Pending the timeout when Stop signal occur
    tonTimeout.IN := FALSE;
END_IF

// Service Process
CASE uiExecutingStep OF
    0:
        // Clear variable
        uiBothStep := 0;
        uiSingleClampStep := 0;
        BoxReady_1st := 0;
        BoxReady_2nd := 0;
        tonTimeOut.IN := FALSE;

        // Check command
        IF M_CheckCommand() THEN
            uiExecutingStep := 10;
        ELSE
            _Error := TRUE;
        END_IF
    10:
        // Start process, check units first
        IF M_CheckUnitsReady() THEN
            uiExecutingStep := 20;
        END_IF
    20:
        // CHeck units not busy state
        IF M_CheckUnitsNotBusy() THEN
            uiExecutingStep := 1000;
        END_IF

    1000:
        // Read   coordinate
        Area := THIS^.Area;
        Address_A := LREAL_TO_INT(Info.A_Position);
        Address_B := LREAL_TO_INT(Info.B_Position);
        DAS_CoreSys.MachineControl.fballocatearea.M_GetPulloutAccess(ControlAccess := E_RoundBeltControlAccess.FanucRobot);

        IF UseA AND NOT UseB THEN
            //Only clampA
            uiExecutingStep := 10000;
        ELSIF NOT UseA AND UseB THEN
            //Only ClampB 
            uiExecutingStep := 20000;
        ELSIF UseA AND UseB THEN
            //Both Clamps
            uiExecutingStep := 30000;
        END_IF

    10000: // Only ClampA 
        IF NOT Robot._DI1.Done THEN

            IF Get THEN // Get box job

                CASE Address_A OF
                    1:
                        DAS_CoreSys.MachineControl.fballocatearea
                            .M_StartStoragePulloutAction(CommandType := E_PullOutConveyorCommandType.SlideB_FeedIn_Ext,
                                                         CV_BackwardTIme := T#0S,
                                                         CV_ForwardTime := T#0S);
                    2:
                        DAS_CoreSys.MachineControl.fballocatearea
                            .M_StartStoragePulloutAction(CommandType := E_PullOutConveyorCommandType.SlideA_FeedIn_Ext,
                                                         CV_BackwardTIme := T#0S,
                                                         CV_ForwardTime := T#0S);
                END_CASE

            ELSE
                CASE Address_A OF
                    1:
                        DAS_CoreSys.MachineControl.fballocatearea
                            .M_StartStoragePulloutAction(CommandType := E_PullOutConveyorCommandType.SlideB_FeedOut_Ext,
                                                         CV_BackwardTIme := T#2S,
                                                         CV_ForwardTime := T#0S);

                    2:
                        DAS_CoreSys.MachineControl.fballocatearea
                            .M_StartStoragePulloutAction(CommandType := E_PullOutConveyorCommandType.SlideA_FeedOut_Ext,
                                                         CV_BackwardTIme := T#2S,
                                                         CV_ForwardTime := T#0S);
                END_CASE

            END_IF

            // Robot Abs move
            Robot.M_StartRobotAbsMove(GetBox := Get,
                                      UseClampA := UseA,
                                      UseClampB := UseB,
                                      Area := Area,
                                      ClampA_Address := Address_A,
                                      ClampB_Address := Address_B,
                                      BoxReady_1 := DAS_CoreSys.MachineControl.fballocatearea.fbPulloutCv.Done,
                                      BoxReady_2 := FALSE);

        ELSE
            tonTimeOut.IN := FALSE;
            uiExecutingStep := 10080;
        END_IF

        IF DAS_CoreSys.MachineControl.fballocatearea.fbPulloutCv.Error THEN
            DAS_CoreSys.MachineControl.fballocatearea.M_StopStoragePulloutAction();
            uiResumeStep := 10000;
            _Abort := TRUE;
            strStatus := 'Feed box error';
        END_IF

        tonTimeOut.IN := TRUE;

        IF tonTimeOut.Q = TRUE THEN
            tonTimeOut.IN := FALSE;
            strStatus := 'Reset Robot timeout';
            _Error := TRUE;
        END_IF
    10080:
        Robot.M_ResetRobotAbsMove(UseA, UseB); // Clear command and go to place box
        DAS_CoreSys.MachineControl.fballocatearea.M_StopStoragePulloutAction();
        tonTimeOut.IN := TRUE;

        IF NOT Robot._DI1.Done THEN
            tonTimeOut.IN := FALSE;
            uiExecutingStep := 99000;
        END_IF

        IF tonTimeOut.Q = TRUE THEN
            strStatus := 'Reset Robot timeout';
            _Error := TRUE;
        END_IF

    20000: // Only ClampB
        IF NOT Robot._DI1.Done THEN

            IF Get THEN // Get box job

                CASE Address_B OF
                    1:
                        DAS_CoreSys.MachineControl.fballocatearea
                            .M_StartStoragePulloutAction(CommandType := E_PullOutConveyorCommandType.SlideB_FeedIn_Ext,
                                                         CV_BackwardTIme := T#2S,
                                                         CV_ForwardTime := T#0S);

                    2:
                        DAS_CoreSys.MachineControl.fballocatearea
                            .M_StartStoragePulloutAction(CommandType := E_PullOutConveyorCommandType.SlideA_FeedIn_Ext,
                                                         CV_BackwardTIme := T#2S,
                                                         CV_ForwardTime := T#0S);
                END_CASE

            ELSE
                CASE Address_B OF
                    1:
                        DAS_CoreSys.MachineControl.fballocatearea
                            .M_StartStoragePulloutAction(CommandType := E_PullOutConveyorCommandType.SlideB_FeedOut_Ext,
                                                         CV_BackwardTIme := T#2S,
                                                         CV_ForwardTime := T#0S);

                    2:
                        DAS_CoreSys.MachineControl.fballocatearea
                            .M_StartStoragePulloutAction(CommandType := E_PullOutConveyorCommandType.SlideA_FeedOut_Ext,
                                                         CV_BackwardTIme := T#2S,
                                                         CV_ForwardTime := T#0S);
                END_CASE

            END_IF

            // Robot Abs move
            Robot.M_StartRobotAbsMove(GetBox := Get,
                                      UseClampA := UseA,
                                      UseClampB := UseB,
                                      Area := Area,
                                      ClampA_Address := Address_A,
                                      ClampB_Address := Address_B,
                                      BoxReady_1 := FALSE,
                                      BoxReady_2 := DAS_CoreSys.MachineControl.fballocatearea.fbPulloutCV.Done);

        ELSE
            tonTimeOut.IN := FALSE;
            uiExecutingStep := 20080;
        END_IF

        IF DAS_CoreSys.MachineControl.fballocatearea.fbPulloutCv.Error THEN
            DAS_CoreSys.MachineControl.fballocatearea.M_StopStoragePulloutAction();
            uiResumeStep := 20000;
            _Abort := TRUE;
            strStatus := 'Feed box timeout';
        END_IF

        tonTimeOut.IN := TRUE;

        IF tonTimeOut.Q = TRUE THEN
            tonTimeOut.IN := FALSE;
            strStatus := 'Reset Robot timeout';
            _Error := TRUE;
        END_IF
    20080:
        Robot.M_ResetRobotAbsMove(UseA, UseB);
        DAS_CoreSys.MachineControl.fballocatearea.M_StopStoragePulloutAction();
        ; // Clear command 

        IF NOT Robot._DI1.Done THEN
            uiExecutingStep := 99000;
        END_IF

        tonTimeOut.IN := TRUE;

        IF tonTimeOut.Q = TRUE THEN
            strStatus := 'Reset Robot timeout';
            _Error := TRUE;
        END_IF
    30000: // Both Clamps

        CASE uiBothStep OF
            0: //	
                BoxReady_1st := FALSE;
                BoxReady_2nd := FALSE;

